REGION Network 1: Khi thang máy ở tầng 1
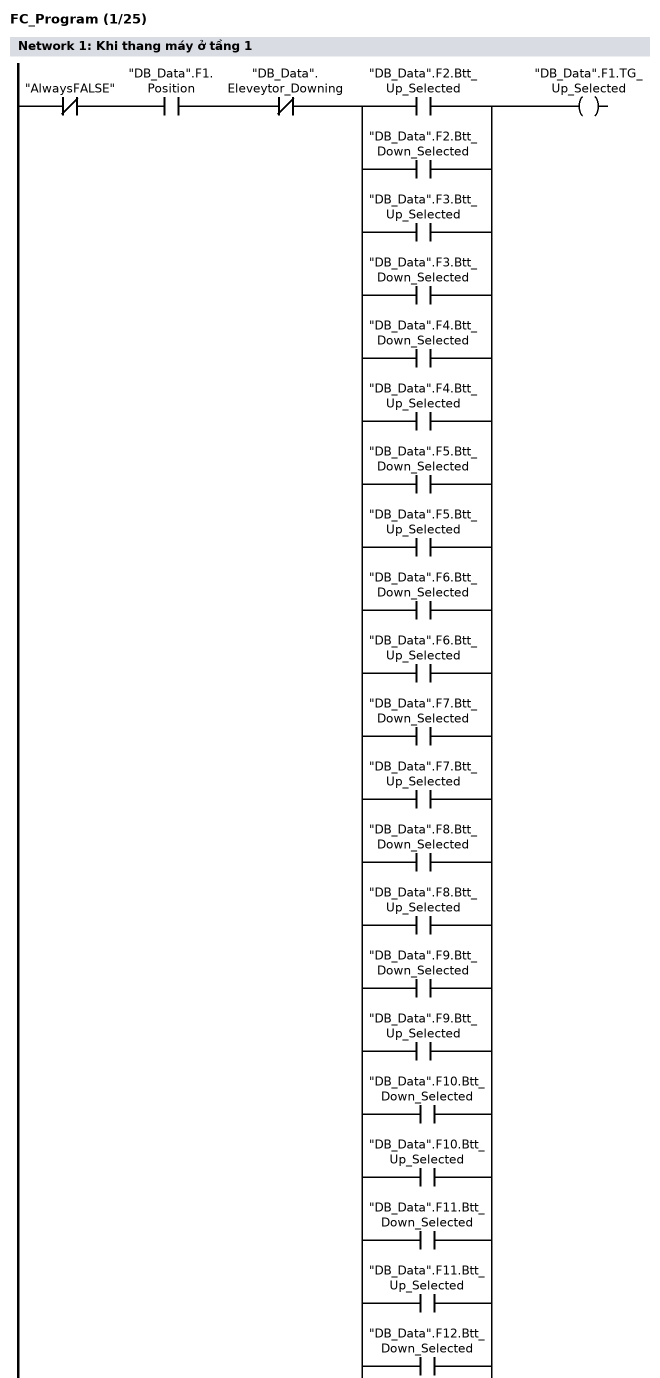
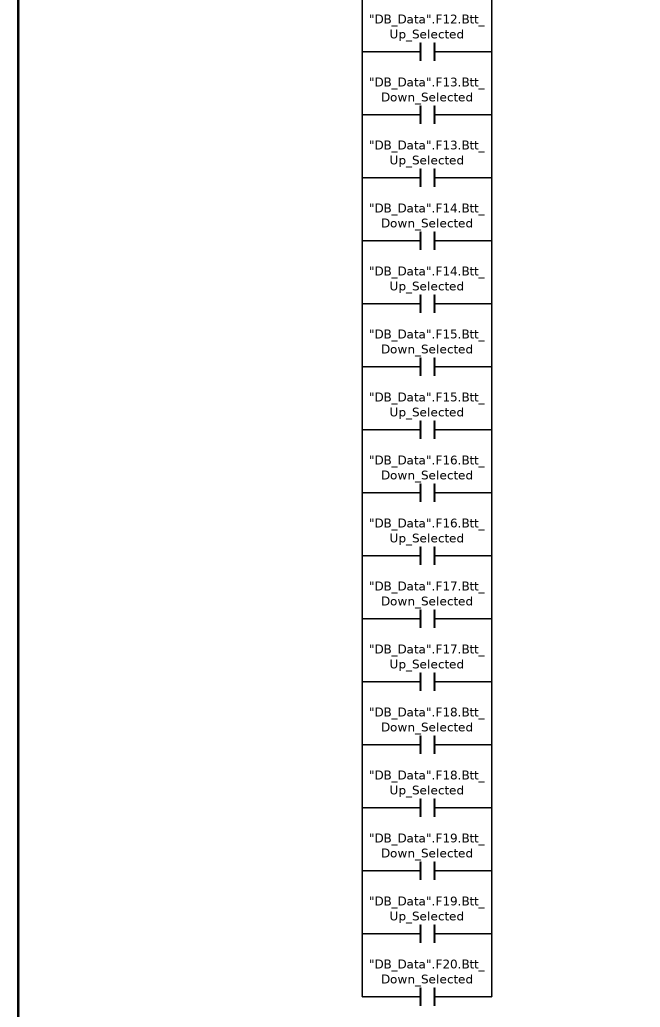
   RUNG wire#powerrail
      I_Contact( "AlwaysFALSE" )
      Contact( "DB_Data".F1.Position )
      I_Contact( "DB_Data".Eleveytor_Downing )
      wire#w1
      Contact( "DB_Data".F2.Btt_Up_Selected )
      wire#w2
      Coil( "DB_Data".F1.TG_Up_Selected )
   END_RUNG
   RUNG wire#w1
      Contact( "DB_Data".F2.Btt_Down_Selected )
   END_RUNG wire#w2
   RUNG wire#w1
      Contact( "DB_Data".F3.Btt_Up_Selected )
   END_RUNG wire#w2
   RUNG wire#w1
      Contact( "DB_Data".F3.Btt_Down_Selected )
   END_RUNG wire#w2
   RUNG wire#w1
      Contact( "DB_Data".F4.Btt_Down_Selected )
   END_RUNG wire#w2
   RUNG wire#w1
      Contact( "DB_Data".F4.Btt_Up_Selected )
   END_RUNG wire#w2
   RUNG wire#w1
      Contact( "DB_Data".F5.Btt_Down_Selected )
   END_RUNG wire#w2
   RUNG wire#w1
      Contact( "DB_Data".F5.Btt_Up_Selected )
   END_RUNG wire#w2
   RUNG wire#w1
      Contact( "DB_Data".F6.Btt_Down_Selected )
   END_RUNG wire#w2
   RUNG wire#w1
      Contact( "DB_Data".F6.Btt_Up_Selected )
   END_RUNG wire#w2
   RUNG wire#w1
      Contact( "DB_Data".F7.Btt_Down_Selected )
   END_RUNG wire#w2
   RUNG wire#w1
      Contact( "DB_Data".F7.Btt_Up_Selected )
   END_RUNG wire#w2
   RUNG wire#w1
      Contact( "DB_Data".F8.Btt_Down_Selected )
   END_RUNG wire#w2
   RUNG wire#w1
      Contact( "DB_Data".F8.Btt_Up_Selected )
   END_RUNG wire#w2
   RUNG wire#w1
      Contact( "DB_Data".F9.Btt_Down_Selected )
   END_RUNG wire#w2
   RUNG wire#w1
      Contact( "DB_Data".F9.Btt_Up_Selected )
   END_RUNG wire#w2
   RUNG wire#w1
      Contact( "DB_Data".F10.Btt_Down_Selected )
   END_RUNG wire#w2
   RUNG wire#w1
      Contact( "DB_Data".F10.Btt_Up_Selected )
   END_RUNG wire#w2
   RUNG wire#w1
      Contact( "DB_Data".F11.Btt_Down_Selected )
   END_RUNG wire#w2
   RUNG wire#w1
      Contact( "DB_Data".F11.Btt_Up_Selected )
   END_RUNG wire#w2
   RUNG wire#w1
      Contact( "DB_Data".F12.Btt_Down_Selected )
   END_RUNG wire#w2
   RUNG wire#w1
      Contact( "DB_Data".F12.Btt_Up_Selected )
   END_RUNG wire#w2
   RUNG wire#w1
      Contact( "DB_Data".F13.Btt_Down_Selected )
   END_RUNG wire#w2
   RUNG wire#w1
      Contact( "DB_Data".F13.Btt_Up_Selected )
   END_RUNG wire#w2
   RUNG wire#w1
      Contact( "DB_Data".F14.Btt_Down_Selected )
   END_RUNG wire#w2
   RUNG wire#w1
      Contact( "DB_Data".F14.Btt_Up_Selected )
   END_RUNG wire#w2
   RUNG wire#w1
      Contact( "DB_Data".F15.Btt_Down_Selected )
   END_RUNG wire#w2
   RUNG wire#w1
      Contact( "DB_Data".F15.Btt_Up_Selected )
   END_RUNG wire#w2
   RUNG wire#w1
      Contact( "DB_Data".F16.Btt_Down_Selected )
   END_RUNG wire#w2
   RUNG wire#w1
      Contact( "DB_Data".F16.Btt_Up_Selected )
   END_RUNG wire#w2
   RUNG wire#w1
      Contact( "DB_Data".F17.Btt_Down_Selected )
   END_RUNG wire#w2
   RUNG wire#w1
      Contact( "DB_Data".F17.Btt_Up_Selected )
   END_RUNG wire#w2
   RUNG wire#w1
      Contact( "DB_Data".F18.Btt_Down_Selected )
   END_RUNG wire#w2
   RUNG wire#w1
      Contact( "DB_Data".F18.Btt_Up_Selected )
   END_RUNG wire#w2
   RUNG wire#w1
      Contact( "DB_Data".F19.Btt_Down_Selected )
   END_RUNG wire#w2
   RUNG wire#w1
      Contact( "DB_Data".F19.Btt_Up_Selected )
   END_RUNG wire#w2
   RUNG wire#w1
      Contact( "DB_Data".F20.Btt_Down_Selected )
   END_RUNG wire#w2
   // the same network as SCL:
   "DB_Data".F1.TG_Up_Selected := NOT "AlwaysFALSE" AND "DB_Data".F1.Position AND NOT "DB_Data".Eleveytor_Downing AND ("DB_Data".F2.Btt_Up_Selected OR "DB_Data".F2.Btt_Down_Selected OR "DB_Data".F3.Btt_Up_Selected OR "DB_Data".F3.Btt_Down_Selected OR "DB_Data".F4.Btt_Down_Selected OR "DB_Data".F4.Btt_Up_Selected OR "DB_Data".F5.Btt_Down_Selected OR "DB_Data".F5.Btt_Up_Selected OR "DB_Data".F6.Btt_Down_Selected OR "DB_Data".F6.Btt_Up_Selected OR "DB_Data".F7.Btt_Down_Selected OR "DB_Data".F7.Btt_Up_Selected OR "DB_Data".F8.Btt_Down_Selected OR "DB_Data".F8.Btt_Up_Selected OR "DB_Data".F9.Btt_Down_Selected OR "DB_Data".F9.Btt_Up_Selected OR "DB_Data".F10.Btt_Down_Selected OR "DB_Data".F10.Btt_Up_Selected OR "DB_Data".F11.Btt_Down_Selected OR "DB_Data".F11.Btt_Up_Selected OR "DB_Data".F12.Btt_Down_Selected OR "DB_Data".F12.Btt_Up_Selected OR "DB_Data".F13.Btt_Down_Selected OR "DB_Data".F13.Btt_Up_Selected OR "DB_Data".F14.Btt_Down_Selected OR "DB_Data".F14.Btt_Up_Selected OR "DB_Data".F15.Btt_Down_Selected OR "DB_Data".F15.Btt_Up_Selected OR "DB_Data".F16.Btt_Down_Selected OR "DB_Data".F16.Btt_Up_Selected OR "DB_Data".F17.Btt_Down_Selected OR "DB_Data".F17.Btt_Up_Selected OR "DB_Data".F18.Btt_Down_Selected OR "DB_Data".F18.Btt_Up_Selected OR "DB_Data".F19.Btt_Down_Selected OR "DB_Data".F19.Btt_Up_Selected OR "DB_Data".F20.Btt_Down_Selected);
END_REGION

REGION Network 2: Khi thang máy ở tầng 2
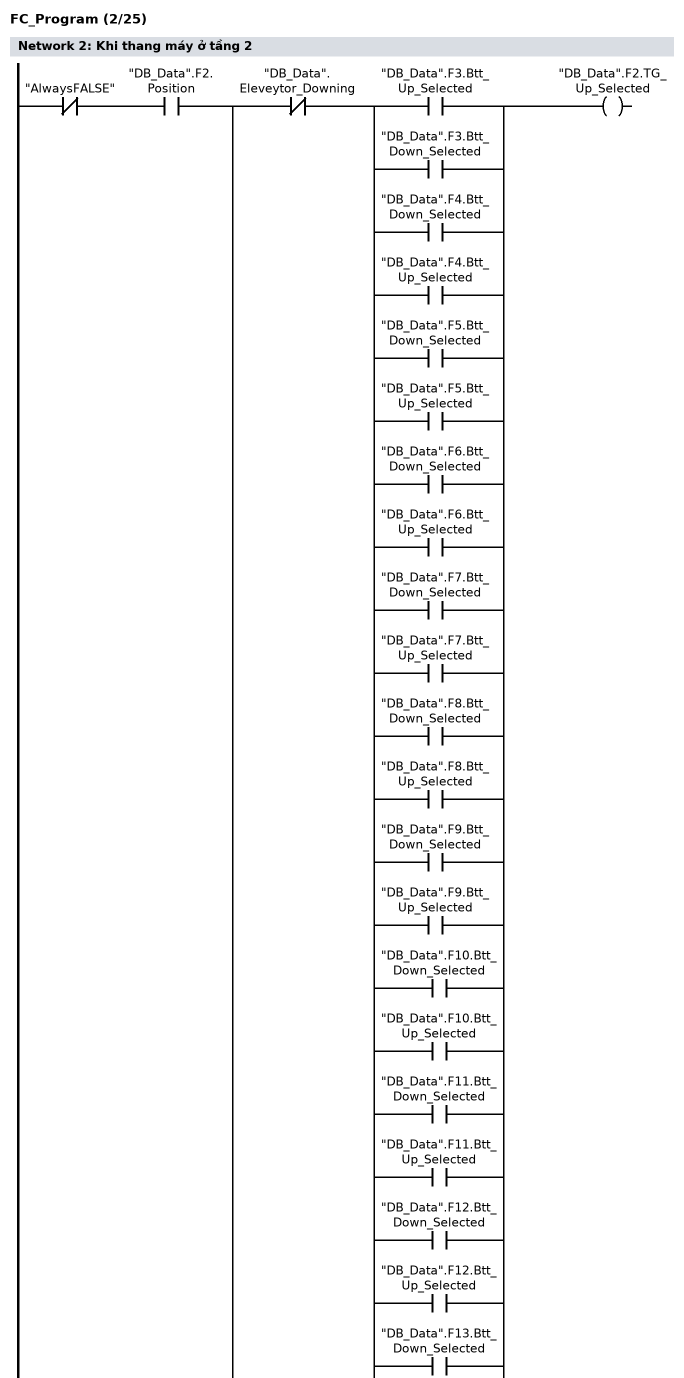
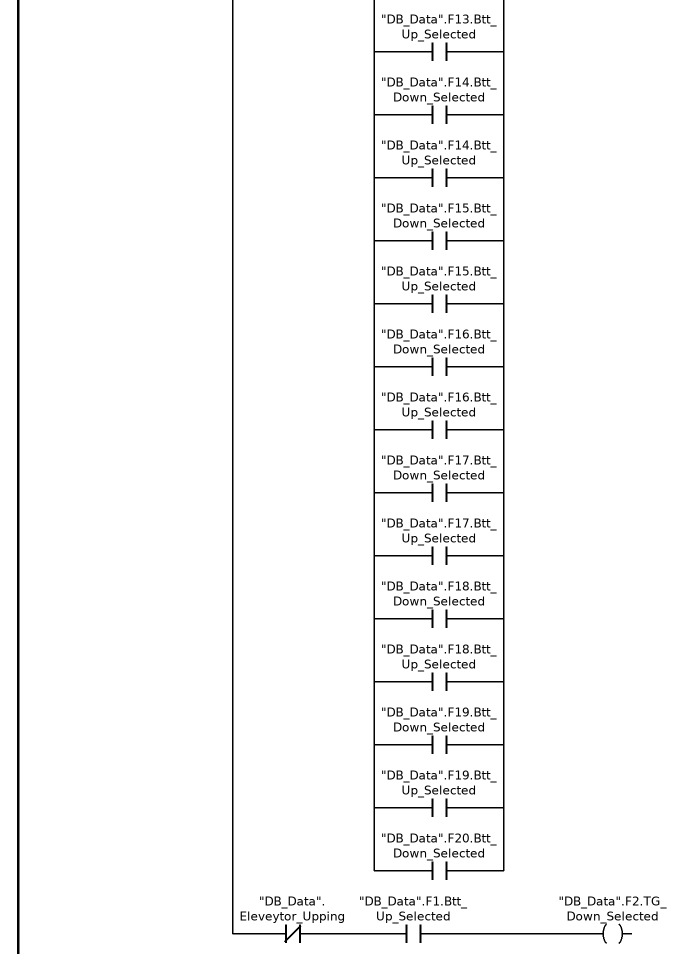
   RUNG wire#powerrail
      I_Contact( "AlwaysFALSE" )
      Contact( "DB_Data".F2.Position )
      wire#w1
      I_Contact( "DB_Data".Eleveytor_Downing )
      wire#w2
      Contact( "DB_Data".F3.Btt_Up_Selected )
      wire#w3
      Coil( "DB_Data".F2.TG_Up_Selected )
   END_RUNG
   RUNG wire#w2
      Contact( "DB_Data".F3.Btt_Down_Selected )
   END_RUNG wire#w3
   RUNG wire#w2
      Contact( "DB_Data".F4.Btt_Down_Selected )
   END_RUNG wire#w3
   RUNG wire#w2
      Contact( "DB_Data".F4.Btt_Up_Selected )
   END_RUNG wire#w3
   RUNG wire#w2
      Contact( "DB_Data".F5.Btt_Down_Selected )
   END_RUNG wire#w3
   RUNG wire#w2
      Contact( "DB_Data".F5.Btt_Up_Selected )
   END_RUNG wire#w3
   RUNG wire#w2
      Contact( "DB_Data".F6.Btt_Down_Selected )
   END_RUNG wire#w3
   RUNG wire#w2
      Contact( "DB_Data".F6.Btt_Up_Selected )
   END_RUNG wire#w3
   RUNG wire#w2
      Contact( "DB_Data".F7.Btt_Down_Selected )
   END_RUNG wire#w3
   RUNG wire#w2
      Contact( "DB_Data".F7.Btt_Up_Selected )
   END_RUNG wire#w3
   RUNG wire#w2
      Contact( "DB_Data".F8.Btt_Down_Selected )
   END_RUNG wire#w3
   RUNG wire#w2
      Contact( "DB_Data".F8.Btt_Up_Selected )
   END_RUNG wire#w3
   RUNG wire#w2
      Contact( "DB_Data".F9.Btt_Down_Selected )
   END_RUNG wire#w3
   RUNG wire#w2
      Contact( "DB_Data".F9.Btt_Up_Selected )
   END_RUNG wire#w3
   RUNG wire#w2
      Contact( "DB_Data".F10.Btt_Down_Selected )
   END_RUNG wire#w3
   RUNG wire#w2
      Contact( "DB_Data".F10.Btt_Up_Selected )
   END_RUNG wire#w3
   RUNG wire#w2
      Contact( "DB_Data".F11.Btt_Down_Selected )
   END_RUNG wire#w3
   RUNG wire#w2
      Contact( "DB_Data".F11.Btt_Up_Selected )
   END_RUNG wire#w3
   RUNG wire#w2
      Contact( "DB_Data".F12.Btt_Down_Selected )
   END_RUNG wire#w3
   RUNG wire#w2
      Contact( "DB_Data".F12.Btt_Up_Selected )
   END_RUNG wire#w3
   RUNG wire#w2
      Contact( "DB_Data".F13.Btt_Down_Selected )
   END_RUNG wire#w3
   RUNG wire#w2
      Contact( "DB_Data".F13.Btt_Up_Selected )
   END_RUNG wire#w3
   RUNG wire#w2
      Contact( "DB_Data".F14.Btt_Down_Selected )
   END_RUNG wire#w3
   RUNG wire#w2
      Contact( "DB_Data".F14.Btt_Up_Selected )
   END_RUNG wire#w3
   RUNG wire#w2
      Contact( "DB_Data".F15.Btt_Down_Selected )
   END_RUNG wire#w3
   RUNG wire#w2
      Contact( "DB_Data".F15.Btt_Up_Selected )
   END_RUNG wire#w3
   RUNG wire#w2
      Contact( "DB_Data".F16.Btt_Down_Selected )
   END_RUNG wire#w3
   RUNG wire#w2
      Contact( "DB_Data".F16.Btt_Up_Selected )
   END_RUNG wire#w3
   RUNG wire#w2
      Contact( "DB_Data".F17.Btt_Down_Selected )
   END_RUNG wire#w3
   RUNG wire#w2
      Contact( "DB_Data".F17.Btt_Up_Selected )
   END_RUNG wire#w3
   RUNG wire#w2
      Contact( "DB_Data".F18.Btt_Down_Selected )
   END_RUNG wire#w3
   RUNG wire#w2
      Contact( "DB_Data".F18.Btt_Up_Selected )
   END_RUNG wire#w3
   RUNG wire#w2
      Contact( "DB_Data".F19.Btt_Down_Selected )
   END_RUNG wire#w3
   RUNG wire#w2
      Contact( "DB_Data".F19.Btt_Up_Selected )
   END_RUNG wire#w3
   RUNG wire#w2
      Contact( "DB_Data".F20.Btt_Down_Selected )
   END_RUNG wire#w3
   RUNG wire#w1
      I_Contact( "DB_Data".Eleveytor_Upping )
      Contact( "DB_Data".F1.Btt_Up_Selected )
      Coil( "DB_Data".F2.TG_Down_Selected )
   END_RUNG
   // the same network as SCL:
   #_w1 := NOT "AlwaysFALSE" AND "DB_Data".F2.Position;
   "DB_Data".F2.TG_Up_Selected := #_w1 AND NOT "DB_Data".Eleveytor_Downing AND ("DB_Data".F3.Btt_Up_Selected OR "DB_Data".F3.Btt_Down_Selected OR "DB_Data".F4.Btt_Down_Selected OR "DB_Data".F4.Btt_Up_Selected OR "DB_Data".F5.Btt_Down_Selected OR "DB_Data".F5.Btt_Up_Selected OR "DB_Data".F6.Btt_Down_Selected OR "DB_Data".F6.Btt_Up_Selected OR "DB_Data".F7.Btt_Down_Selected OR "DB_Data".F7.Btt_Up_Selected OR "DB_Data".F8.Btt_Down_Selected OR "DB_Data".F8.Btt_Up_Selected OR "DB_Data".F9.Btt_Down_Selected OR "DB_Data".F9.Btt_Up_Selected OR "DB_Data".F10.Btt_Down_Selected OR "DB_Data".F10.Btt_Up_Selected OR "DB_Data".F11.Btt_Down_Selected OR "DB_Data".F11.Btt_Up_Selected OR "DB_Data".F12.Btt_Down_Selected OR "DB_Data".F12.Btt_Up_Selected OR "DB_Data".F13.Btt_Down_Selected OR "DB_Data".F13.Btt_Up_Selected OR "DB_Data".F14.Btt_Down_Selected OR "DB_Data".F14.Btt_Up_Selected OR "DB_Data".F15.Btt_Down_Selected OR "DB_Data".F15.Btt_Up_Selected OR "DB_Data".F16.Btt_Down_Selected OR "DB_Data".F16.Btt_Up_Selected OR "DB_Data".F17.Btt_Down_Selected OR "DB_Data".F17.Btt_Up_Selected OR "DB_Data".F18.Btt_Down_Selected OR "DB_Data".F18.Btt_Up_Selected OR "DB_Data".F19.Btt_Down_Selected OR "DB_Data".F19.Btt_Up_Selected OR "DB_Data".F20.Btt_Down_Selected);
   "DB_Data".F2.TG_Down_Selected := #_w1 AND NOT "DB_Data".Eleveytor_Upping AND "DB_Data".F1.Btt_Up_Selected;
END_REGION

REGION Network 3: Khi thang máy ở tầng 3
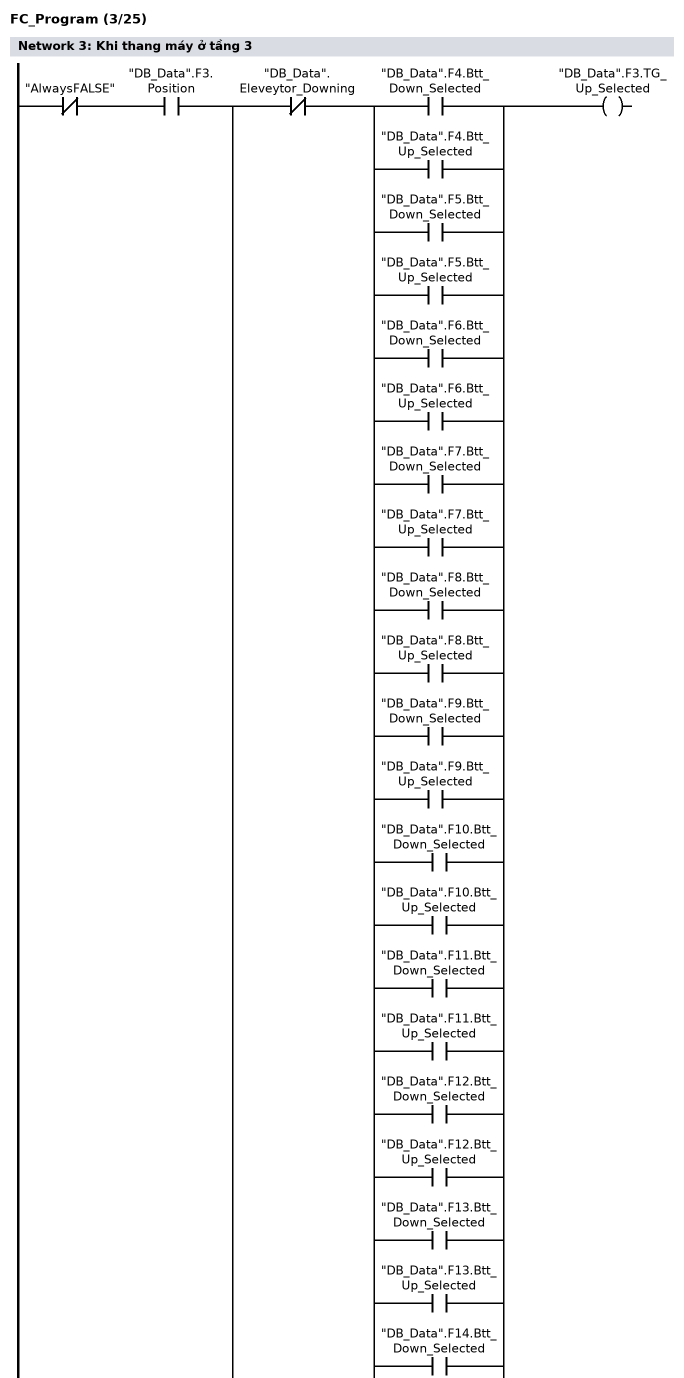
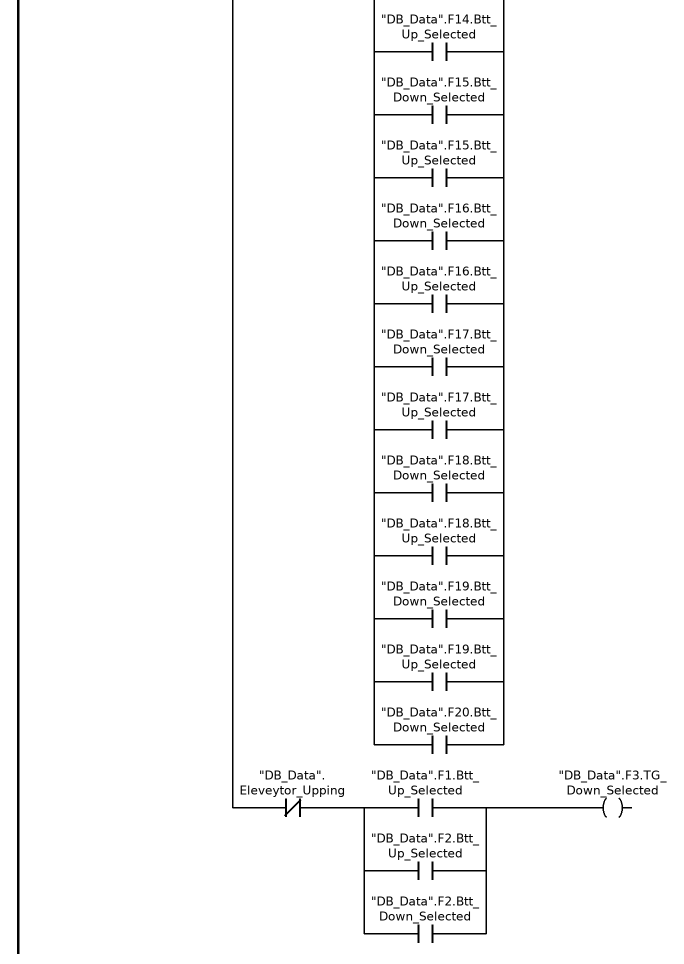
   RUNG wire#powerrail
      I_Contact( "AlwaysFALSE" )
      Contact( "DB_Data".F3.Position )
      wire#w1
      I_Contact( "DB_Data".Eleveytor_Downing )
      wire#w2
      Contact( "DB_Data".F4.Btt_Down_Selected )
      wire#w3
      Coil( "DB_Data".F3.TG_Up_Selected )
   END_RUNG
   RUNG wire#w2
      Contact( "DB_Data".F4.Btt_Up_Selected )
   END_RUNG wire#w3
   RUNG wire#w2
      Contact( "DB_Data".F5.Btt_Down_Selected )
   END_RUNG wire#w3
   RUNG wire#w2
      Contact( "DB_Data".F5.Btt_Up_Selected )
   END_RUNG wire#w3
   RUNG wire#w2
      Contact( "DB_Data".F6.Btt_Down_Selected )
   END_RUNG wire#w3
   RUNG wire#w2
      Contact( "DB_Data".F6.Btt_Up_Selected )
   END_RUNG wire#w3
   RUNG wire#w2
      Contact( "DB_Data".F7.Btt_Down_Selected )
   END_RUNG wire#w3
   RUNG wire#w2
      Contact( "DB_Data".F7.Btt_Up_Selected )
   END_RUNG wire#w3
   RUNG wire#w2
      Contact( "DB_Data".F8.Btt_Down_Selected )
   END_RUNG wire#w3
   RUNG wire#w2
      Contact( "DB_Data".F8.Btt_Up_Selected )
   END_RUNG wire#w3
   RUNG wire#w2
      Contact( "DB_Data".F9.Btt_Down_Selected )
   END_RUNG wire#w3
   RUNG wire#w2
      Contact( "DB_Data".F9.Btt_Up_Selected )
   END_RUNG wire#w3
   RUNG wire#w2
      Contact( "DB_Data".F10.Btt_Down_Selected )
   END_RUNG wire#w3
   RUNG wire#w2
      Contact( "DB_Data".F10.Btt_Up_Selected )
   END_RUNG wire#w3
   RUNG wire#w2
      Contact( "DB_Data".F11.Btt_Down_Selected )
   END_RUNG wire#w3
   RUNG wire#w2
      Contact( "DB_Data".F11.Btt_Up_Selected )
   END_RUNG wire#w3
   RUNG wire#w2
      Contact( "DB_Data".F12.Btt_Down_Selected )
   END_RUNG wire#w3
   RUNG wire#w2
      Contact( "DB_Data".F12.Btt_Up_Selected )
   END_RUNG wire#w3
   RUNG wire#w2
      Contact( "DB_Data".F13.Btt_Down_Selected )
   END_RUNG wire#w3
   RUNG wire#w2
      Contact( "DB_Data".F13.Btt_Up_Selected )
   END_RUNG wire#w3
   RUNG wire#w2
      Contact( "DB_Data".F14.Btt_Down_Selected )
   END_RUNG wire#w3
   RUNG wire#w2
      Contact( "DB_Data".F14.Btt_Up_Selected )
   END_RUNG wire#w3
   RUNG wire#w2
      Contact( "DB_Data".F15.Btt_Down_Selected )
   END_RUNG wire#w3
   RUNG wire#w2
      Contact( "DB_Data".F15.Btt_Up_Selected )
   END_RUNG wire#w3
   RUNG wire#w2
      Contact( "DB_Data".F16.Btt_Down_Selected )
   END_RUNG wire#w3
   RUNG wire#w2
      Contact( "DB_Data".F16.Btt_Up_Selected )
   END_RUNG wire#w3
   RUNG wire#w2
      Contact( "DB_Data".F17.Btt_Down_Selected )
   END_RUNG wire#w3
   RUNG wire#w2
      Contact( "DB_Data".F17.Btt_Up_Selected )
   END_RUNG wire#w3
   RUNG wire#w2
      Contact( "DB_Data".F18.Btt_Down_Selected )
   END_RUNG wire#w3
   RUNG wire#w2
      Contact( "DB_Data".F18.Btt_Up_Selected )
   END_RUNG wire#w3
   RUNG wire#w2
      Contact( "DB_Data".F19.Btt_Down_Selected )
   END_RUNG wire#w3
   RUNG wire#w2
      Contact( "DB_Data".F19.Btt_Up_Selected )
   END_RUNG wire#w3
   RUNG wire#w2
      Contact( "DB_Data".F20.Btt_Down_Selected )
   END_RUNG wire#w3
   RUNG wire#w1
      I_Contact( "DB_Data".Eleveytor_Upping )
      wire#w4
      Contact( "DB_Data".F1.Btt_Up_Selected )
      wire#w5
      Coil( "DB_Data".F3.TG_Down_Selected )
   END_RUNG
   RUNG wire#w4
      Contact( "DB_Data".F2.Btt_Up_Selected )
   END_RUNG wire#w5
   RUNG wire#w4
      Contact( "DB_Data".F2.Btt_Down_Selected )
   END_RUNG wire#w5
   // the same network as SCL:
   #_w1 := NOT "AlwaysFALSE" AND "DB_Data".F3.Position;
   "DB_Data".F3.TG_Up_Selected := #_w1 AND NOT "DB_Data".Eleveytor_Downing AND ("DB_Data".F4.Btt_Down_Selected OR "DB_Data".F4.Btt_Up_Selected OR "DB_Data".F5.Btt_Down_Selected OR "DB_Data".F5.Btt_Up_Selected OR "DB_Data".F6.Btt_Down_Selected OR "DB_Data".F6.Btt_Up_Selected OR "DB_Data".F7.Btt_Down_Selected OR "DB_Data".F7.Btt_Up_Selected OR "DB_Data".F8.Btt_Down_Selected OR "DB_Data".F8.Btt_Up_Selected OR "DB_Data".F9.Btt_Down_Selected OR "DB_Data".F9.Btt_Up_Selected OR "DB_Data".F10.Btt_Down_Selected OR "DB_Data".F10.Btt_Up_Selected OR "DB_Data".F11.Btt_Down_Selected OR "DB_Data".F11.Btt_Up_Selected OR "DB_Data".F12.Btt_Down_Selected OR "DB_Data".F12.Btt_Up_Selected OR "DB_Data".F13.Btt_Down_Selected OR "DB_Data".F13.Btt_Up_Selected OR "DB_Data".F14.Btt_Down_Selected OR "DB_Data".F14.Btt_Up_Selected OR "DB_Data".F15.Btt_Down_Selected OR "DB_Data".F15.Btt_Up_Selected OR "DB_Data".F16.Btt_Down_Selected OR "DB_Data".F16.Btt_Up_Selected OR "DB_Data".F17.Btt_Down_Selected OR "DB_Data".F17.Btt_Up_Selected OR "DB_Data".F18.Btt_Down_Selected OR "DB_Data".F18.Btt_Up_Selected OR "DB_Data".F19.Btt_Down_Selected OR "DB_Data".F19.Btt_Up_Selected OR "DB_Data".F20.Btt_Down_Selected);
   "DB_Data".F3.TG_Down_Selected := #_w1 AND NOT "DB_Data".Eleveytor_Upping AND ("DB_Data".F1.Btt_Up_Selected OR "DB_Data".F2.Btt_Up_Selected OR "DB_Data".F2.Btt_Down_Selected);
END_REGION

REGION Network 4: Khi thang máy ở tầng 4
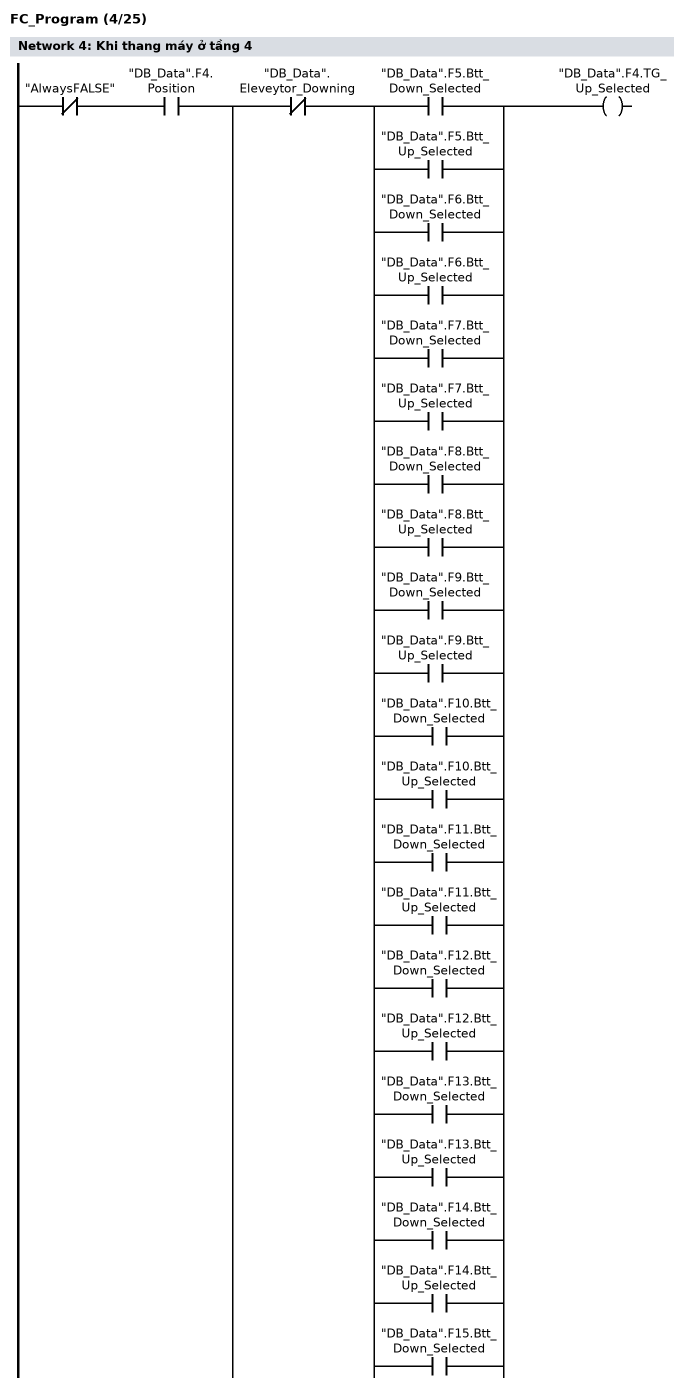
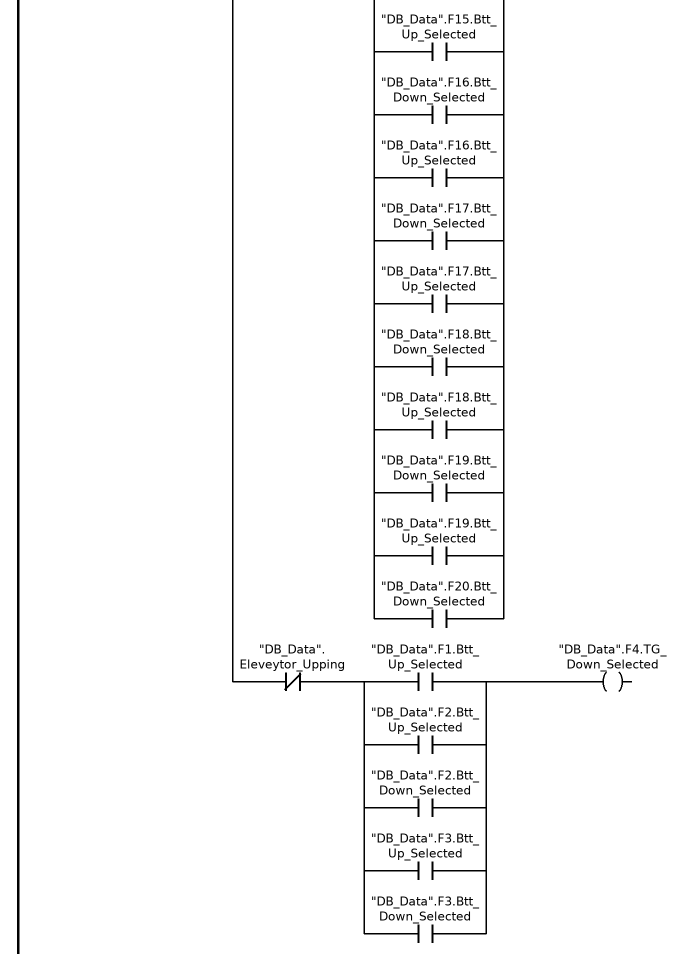
   RUNG wire#powerrail
      I_Contact( "AlwaysFALSE" )
      Contact( "DB_Data".F4.Position )
      wire#w1
      I_Contact( "DB_Data".Eleveytor_Downing )
      wire#w2
      Contact( "DB_Data".F5.Btt_Down_Selected )
      wire#w3
      Coil( "DB_Data".F4.TG_Up_Selected )
   END_RUNG
   RUNG wire#w2
      Contact( "DB_Data".F5.Btt_Up_Selected )
   END_RUNG wire#w3
   RUNG wire#w2
      Contact( "DB_Data".F6.Btt_Down_Selected )
   END_RUNG wire#w3
   RUNG wire#w2
      Contact( "DB_Data".F6.Btt_Up_Selected )
   END_RUNG wire#w3
   RUNG wire#w2
      Contact( "DB_Data".F7.Btt_Down_Selected )
   END_RUNG wire#w3
   RUNG wire#w2
      Contact( "DB_Data".F7.Btt_Up_Selected )
   END_RUNG wire#w3
   RUNG wire#w2
      Contact( "DB_Data".F8.Btt_Down_Selected )
   END_RUNG wire#w3
   RUNG wire#w2
      Contact( "DB_Data".F8.Btt_Up_Selected )
   END_RUNG wire#w3
   RUNG wire#w2
      Contact( "DB_Data".F9.Btt_Down_Selected )
   END_RUNG wire#w3
   RUNG wire#w2
      Contact( "DB_Data".F9.Btt_Up_Selected )
   END_RUNG wire#w3
   RUNG wire#w2
      Contact( "DB_Data".F10.Btt_Down_Selected )
   END_RUNG wire#w3
   RUNG wire#w2
      Contact( "DB_Data".F10.Btt_Up_Selected )
   END_RUNG wire#w3
   RUNG wire#w2
      Contact( "DB_Data".F11.Btt_Down_Selected )
   END_RUNG wire#w3
   RUNG wire#w2
      Contact( "DB_Data".F11.Btt_Up_Selected )
   END_RUNG wire#w3
   RUNG wire#w2
      Contact( "DB_Data".F12.Btt_Down_Selected )
   END_RUNG wire#w3
   RUNG wire#w2
      Contact( "DB_Data".F12.Btt_Up_Selected )
   END_RUNG wire#w3
   RUNG wire#w2
      Contact( "DB_Data".F13.Btt_Down_Selected )
   END_RUNG wire#w3
   RUNG wire#w2
      Contact( "DB_Data".F13.Btt_Up_Selected )
   END_RUNG wire#w3
   RUNG wire#w2
      Contact( "DB_Data".F14.Btt_Down_Selected )
   END_RUNG wire#w3
   RUNG wire#w2
      Contact( "DB_Data".F14.Btt_Up_Selected )
   END_RUNG wire#w3
   RUNG wire#w2
      Contact( "DB_Data".F15.Btt_Down_Selected )
   END_RUNG wire#w3
   RUNG wire#w2
      Contact( "DB_Data".F15.Btt_Up_Selected )
   END_RUNG wire#w3
   RUNG wire#w2
      Contact( "DB_Data".F16.Btt_Down_Selected )
   END_RUNG wire#w3
   RUNG wire#w2
      Contact( "DB_Data".F16.Btt_Up_Selected )
   END_RUNG wire#w3
   RUNG wire#w2
      Contact( "DB_Data".F17.Btt_Down_Selected )
   END_RUNG wire#w3
   RUNG wire#w2
      Contact( "DB_Data".F17.Btt_Up_Selected )
   END_RUNG wire#w3
   RUNG wire#w2
      Contact( "DB_Data".F18.Btt_Down_Selected )
   END_RUNG wire#w3
   RUNG wire#w2
      Contact( "DB_Data".F18.Btt_Up_Selected )
   END_RUNG wire#w3
   RUNG wire#w2
      Contact( "DB_Data".F19.Btt_Down_Selected )
   END_RUNG wire#w3
   RUNG wire#w2
      Contact( "DB_Data".F19.Btt_Up_Selected )
   END_RUNG wire#w3
   RUNG wire#w2
      Contact( "DB_Data".F20.Btt_Down_Selected )
   END_RUNG wire#w3
   RUNG wire#w1
      I_Contact( "DB_Data".Eleveytor_Upping )
      wire#w4
      Contact( "DB_Data".F1.Btt_Up_Selected )
      wire#w5
      Coil( "DB_Data".F4.TG_Down_Selected )
   END_RUNG
   RUNG wire#w4
      Contact( "DB_Data".F2.Btt_Up_Selected )
   END_RUNG wire#w5
   RUNG wire#w4
      Contact( "DB_Data".F2.Btt_Down_Selected )
   END_RUNG wire#w5
   RUNG wire#w4
      Contact( "DB_Data".F3.Btt_Up_Selected )
   END_RUNG wire#w5
   RUNG wire#w4
      Contact( "DB_Data".F3.Btt_Down_Selected )
   END_RUNG wire#w5
   // the same network as SCL:
   #_w1 := NOT "AlwaysFALSE" AND "DB_Data".F4.Position;
   "DB_Data".F4.TG_Up_Selected := #_w1 AND NOT "DB_Data".Eleveytor_Downing AND ("DB_Data".F5.Btt_Down_Selected OR "DB_Data".F5.Btt_Up_Selected OR "DB_Data".F6.Btt_Down_Selected OR "DB_Data".F6.Btt_Up_Selected OR "DB_Data".F7.Btt_Down_Selected OR "DB_Data".F7.Btt_Up_Selected OR "DB_Data".F8.Btt_Down_Selected OR "DB_Data".F8.Btt_Up_Selected OR "DB_Data".F9.Btt_Down_Selected OR "DB_Data".F9.Btt_Up_Selected OR "DB_Data".F10.Btt_Down_Selected OR "DB_Data".F10.Btt_Up_Selected OR "DB_Data".F11.Btt_Down_Selected OR "DB_Data".F11.Btt_Up_Selected OR "DB_Data".F12.Btt_Down_Selected OR "DB_Data".F12.Btt_Up_Selected OR "DB_Data".F13.Btt_Down_Selected OR "DB_Data".F13.Btt_Up_Selected OR "DB_Data".F14.Btt_Down_Selected OR "DB_Data".F14.Btt_Up_Selected OR "DB_Data".F15.Btt_Down_Selected OR "DB_Data".F15.Btt_Up_Selected OR "DB_Data".F16.Btt_Down_Selected OR "DB_Data".F16.Btt_Up_Selected OR "DB_Data".F17.Btt_Down_Selected OR "DB_Data".F17.Btt_Up_Selected OR "DB_Data".F18.Btt_Down_Selected OR "DB_Data".F18.Btt_Up_Selected OR "DB_Data".F19.Btt_Down_Selected OR "DB_Data".F19.Btt_Up_Selected OR "DB_Data".F20.Btt_Down_Selected);
   "DB_Data".F4.TG_Down_Selected := #_w1 AND NOT "DB_Data".Eleveytor_Upping AND ("DB_Data".F1.Btt_Up_Selected OR "DB_Data".F2.Btt_Up_Selected OR "DB_Data".F2.Btt_Down_Selected OR "DB_Data".F3.Btt_Up_Selected OR "DB_Data".F3.Btt_Down_Selected);
END_REGION

REGION Network 5: Khi thang máy ở tầng 5
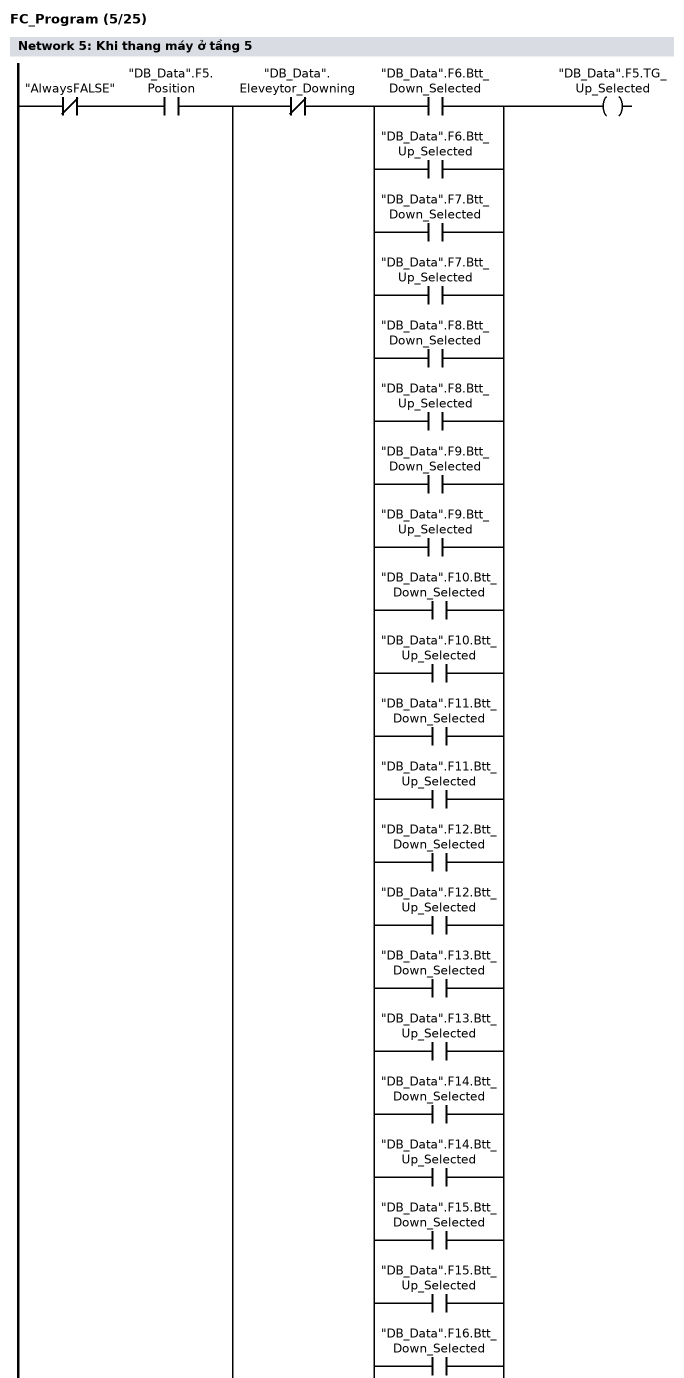
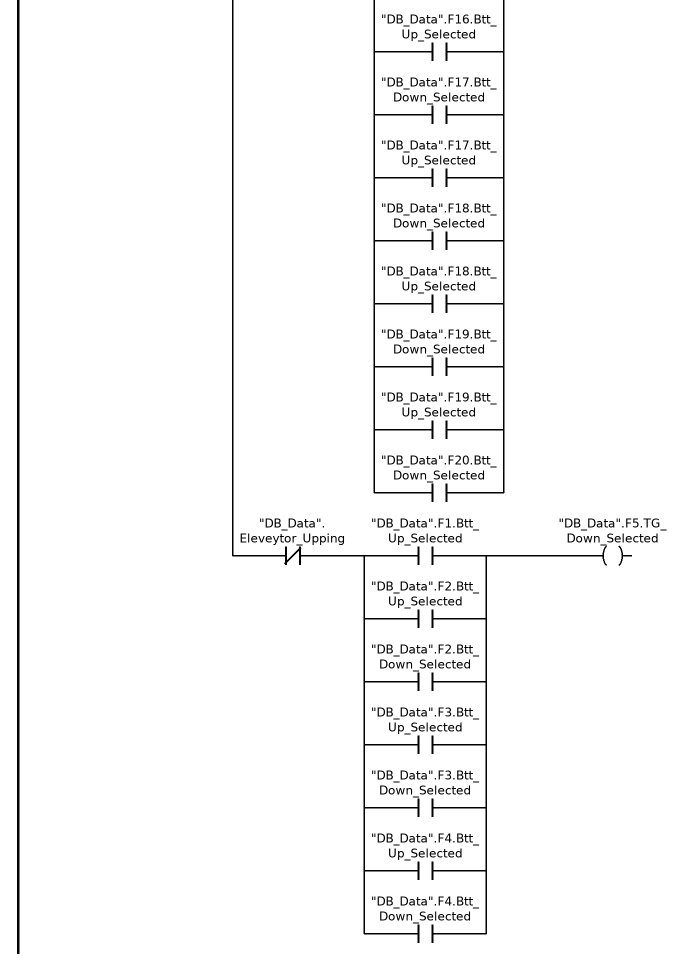
   RUNG wire#powerrail
      I_Contact( "AlwaysFALSE" )
      Contact( "DB_Data".F5.Position )
      wire#w1
      I_Contact( "DB_Data".Eleveytor_Downing )
      wire#w2
      Contact( "DB_Data".F6.Btt_Down_Selected )
      wire#w3
      Coil( "DB_Data".F5.TG_Up_Selected )
   END_RUNG
   RUNG wire#w2
      Contact( "DB_Data".F6.Btt_Up_Selected )
   END_RUNG wire#w3
   RUNG wire#w2
      Contact( "DB_Data".F7.Btt_Down_Selected )
   END_RUNG wire#w3
   RUNG wire#w2
      Contact( "DB_Data".F7.Btt_Up_Selected )
   END_RUNG wire#w3
   RUNG wire#w2
      Contact( "DB_Data".F8.Btt_Down_Selected )
   END_RUNG wire#w3
   RUNG wire#w2
      Contact( "DB_Data".F8.Btt_Up_Selected )
   END_RUNG wire#w3
   RUNG wire#w2
      Contact( "DB_Data".F9.Btt_Down_Selected )
   END_RUNG wire#w3
   RUNG wire#w2
      Contact( "DB_Data".F9.Btt_Up_Selected )
   END_RUNG wire#w3
   RUNG wire#w2
      Contact( "DB_Data".F10.Btt_Down_Selected )
   END_RUNG wire#w3
   RUNG wire#w2
      Contact( "DB_Data".F10.Btt_Up_Selected )
   END_RUNG wire#w3
   RUNG wire#w2
      Contact( "DB_Data".F11.Btt_Down_Selected )
   END_RUNG wire#w3
   RUNG wire#w2
      Contact( "DB_Data".F11.Btt_Up_Selected )
   END_RUNG wire#w3
   RUNG wire#w2
      Contact( "DB_Data".F12.Btt_Down_Selected )
   END_RUNG wire#w3
   RUNG wire#w2
      Contact( "DB_Data".F12.Btt_Up_Selected )
   END_RUNG wire#w3
   RUNG wire#w2
      Contact( "DB_Data".F13.Btt_Down_Selected )
   END_RUNG wire#w3
   RUNG wire#w2
      Contact( "DB_Data".F13.Btt_Up_Selected )
   END_RUNG wire#w3
   RUNG wire#w2
      Contact( "DB_Data".F14.Btt_Down_Selected )
   END_RUNG wire#w3
   RUNG wire#w2
      Contact( "DB_Data".F14.Btt_Up_Selected )
   END_RUNG wire#w3
   RUNG wire#w2
      Contact( "DB_Data".F15.Btt_Down_Selected )
   END_RUNG wire#w3
   RUNG wire#w2
      Contact( "DB_Data".F15.Btt_Up_Selected )
   END_RUNG wire#w3
   RUNG wire#w2
      Contact( "DB_Data".F16.Btt_Down_Selected )
   END_RUNG wire#w3
   RUNG wire#w2
      Contact( "DB_Data".F16.Btt_Up_Selected )
   END_RUNG wire#w3
   RUNG wire#w2
      Contact( "DB_Data".F17.Btt_Down_Selected )
   END_RUNG wire#w3
   RUNG wire#w2
      Contact( "DB_Data".F17.Btt_Up_Selected )
   END_RUNG wire#w3
   RUNG wire#w2
      Contact( "DB_Data".F18.Btt_Down_Selected )
   END_RUNG wire#w3
   RUNG wire#w2
      Contact( "DB_Data".F18.Btt_Up_Selected )
   END_RUNG wire#w3
   RUNG wire#w2
      Contact( "DB_Data".F19.Btt_Down_Selected )
   END_RUNG wire#w3
   RUNG wire#w2
      Contact( "DB_Data".F19.Btt_Up_Selected )
   END_RUNG wire#w3
   RUNG wire#w2
      Contact( "DB_Data".F20.Btt_Down_Selected )
   END_RUNG wire#w3
   RUNG wire#w1
      I_Contact( "DB_Data".Eleveytor_Upping )
      wire#w4
      Contact( "DB_Data".F1.Btt_Up_Selected )
      wire#w5
      Coil( "DB_Data".F5.TG_Down_Selected )
   END_RUNG
   RUNG wire#w4
      Contact( "DB_Data".F2.Btt_Up_Selected )
   END_RUNG wire#w5
   RUNG wire#w4
      Contact( "DB_Data".F2.Btt_Down_Selected )
   END_RUNG wire#w5
   RUNG wire#w4
      Contact( "DB_Data".F3.Btt_Up_Selected )
   END_RUNG wire#w5
   RUNG wire#w4
      Contact( "DB_Data".F3.Btt_Down_Selected )
   END_RUNG wire#w5
   RUNG wire#w4
      Contact( "DB_Data".F4.Btt_Up_Selected )
   END_RUNG wire#w5
   RUNG wire#w4
      Contact( "DB_Data".F4.Btt_Down_Selected )
   END_RUNG wire#w5
   // the same network as SCL:
   #_w1 := NOT "AlwaysFALSE" AND "DB_Data".F5.Position;
   "DB_Data".F5.TG_Up_Selected := #_w1 AND NOT "DB_Data".Eleveytor_Downing AND ("DB_Data".F6.Btt_Down_Selected OR "DB_Data".F6.Btt_Up_Selected OR "DB_Data".F7.Btt_Down_Selected OR "DB_Data".F7.Btt_Up_Selected OR "DB_Data".F8.Btt_Down_Selected OR "DB_Data".F8.Btt_Up_Selected OR "DB_Data".F9.Btt_Down_Selected OR "DB_Data".F9.Btt_Up_Selected OR "DB_Data".F10.Btt_Down_Selected OR "DB_Data".F10.Btt_Up_Selected OR "DB_Data".F11.Btt_Down_Selected OR "DB_Data".F11.Btt_Up_Selected OR "DB_Data".F12.Btt_Down_Selected OR "DB_Data".F12.Btt_Up_Selected OR "DB_Data".F13.Btt_Down_Selected OR "DB_Data".F13.Btt_Up_Selected OR "DB_Data".F14.Btt_Down_Selected OR "DB_Data".F14.Btt_Up_Selected OR "DB_Data".F15.Btt_Down_Selected OR "DB_Data".F15.Btt_Up_Selected OR "DB_Data".F16.Btt_Down_Selected OR "DB_Data".F16.Btt_Up_Selected OR "DB_Data".F17.Btt_Down_Selected OR "DB_Data".F17.Btt_Up_Selected OR "DB_Data".F18.Btt_Down_Selected OR "DB_Data".F18.Btt_Up_Selected OR "DB_Data".F19.Btt_Down_Selected OR "DB_Data".F19.Btt_Up_Selected OR "DB_Data".F20.Btt_Down_Selected);
   "DB_Data".F5.TG_Down_Selected := #_w1 AND NOT "DB_Data".Eleveytor_Upping AND ("DB_Data".F1.Btt_Up_Selected OR "DB_Data".F2.Btt_Up_Selected OR "DB_Data".F2.Btt_Down_Selected OR "DB_Data".F3.Btt_Up_Selected OR "DB_Data".F3.Btt_Down_Selected OR "DB_Data".F4.Btt_Up_Selected OR "DB_Data".F4.Btt_Down_Selected);
END_REGION

REGION Network 6: Khi thang máy ở tầng 6
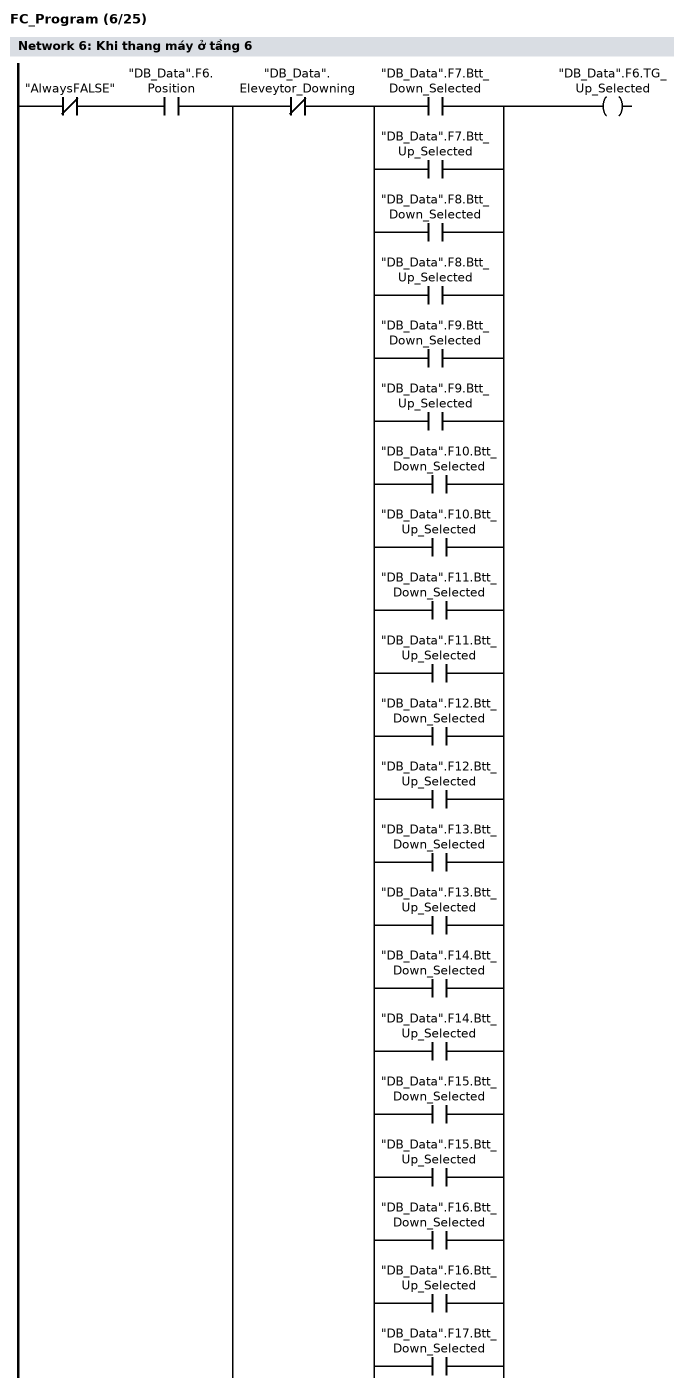
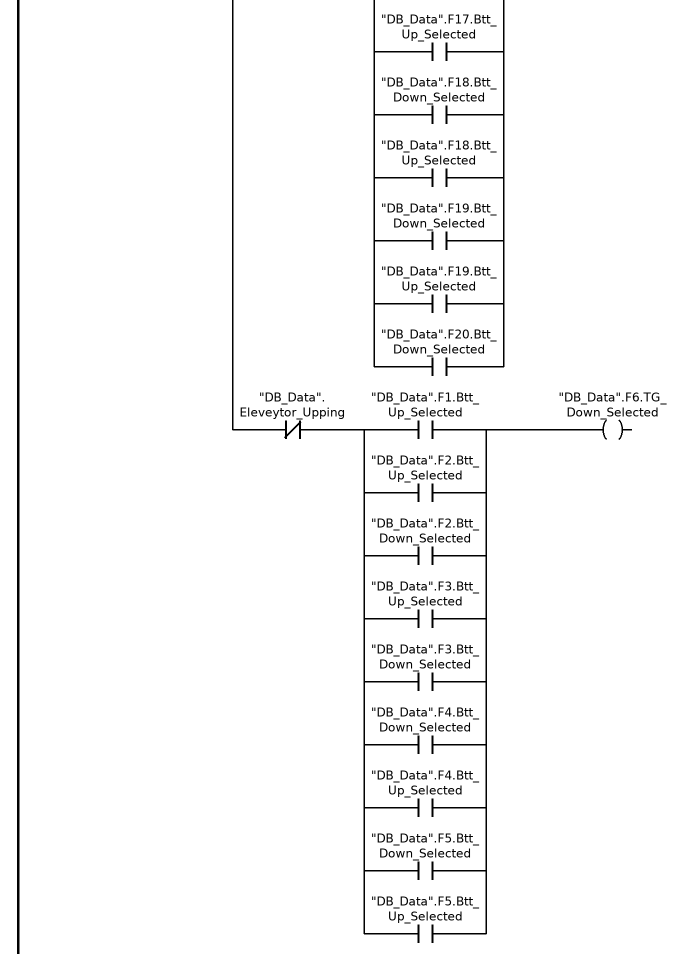
   RUNG wire#powerrail
      I_Contact( "AlwaysFALSE" )
      Contact( "DB_Data".F6.Position )
      wire#w1
      I_Contact( "DB_Data".Eleveytor_Downing )
      wire#w2
      Contact( "DB_Data".F7.Btt_Down_Selected )
      wire#w3
      Coil( "DB_Data".F6.TG_Up_Selected )
   END_RUNG
   RUNG wire#w2
      Contact( "DB_Data".F7.Btt_Up_Selected )
   END_RUNG wire#w3
   RUNG wire#w2
      Contact( "DB_Data".F8.Btt_Down_Selected )
   END_RUNG wire#w3
   RUNG wire#w2
      Contact( "DB_Data".F8.Btt_Up_Selected )
   END_RUNG wire#w3
   RUNG wire#w2
      Contact( "DB_Data".F9.Btt_Down_Selected )
   END_RUNG wire#w3
   RUNG wire#w2
      Contact( "DB_Data".F9.Btt_Up_Selected )
   END_RUNG wire#w3
   RUNG wire#w2
      Contact( "DB_Data".F10.Btt_Down_Selected )
   END_RUNG wire#w3
   RUNG wire#w2
      Contact( "DB_Data".F10.Btt_Up_Selected )
   END_RUNG wire#w3
   RUNG wire#w2
      Contact( "DB_Data".F11.Btt_Down_Selected )
   END_RUNG wire#w3
   RUNG wire#w2
      Contact( "DB_Data".F11.Btt_Up_Selected )
   END_RUNG wire#w3
   RUNG wire#w2
      Contact( "DB_Data".F12.Btt_Down_Selected )
   END_RUNG wire#w3
   RUNG wire#w2
      Contact( "DB_Data".F12.Btt_Up_Selected )
   END_RUNG wire#w3
   RUNG wire#w2
      Contact( "DB_Data".F13.Btt_Down_Selected )
   END_RUNG wire#w3
   RUNG wire#w2
      Contact( "DB_Data".F13.Btt_Up_Selected )
   END_RUNG wire#w3
   RUNG wire#w2
      Contact( "DB_Data".F14.Btt_Down_Selected )
   END_RUNG wire#w3
   RUNG wire#w2
      Contact( "DB_Data".F14.Btt_Up_Selected )
   END_RUNG wire#w3
   RUNG wire#w2
      Contact( "DB_Data".F15.Btt_Down_Selected )
   END_RUNG wire#w3
   RUNG wire#w2
      Contact( "DB_Data".F15.Btt_Up_Selected )
   END_RUNG wire#w3
   RUNG wire#w2
      Contact( "DB_Data".F16.Btt_Down_Selected )
   END_RUNG wire#w3
   RUNG wire#w2
      Contact( "DB_Data".F16.Btt_Up_Selected )
   END_RUNG wire#w3
   RUNG wire#w2
      Contact( "DB_Data".F17.Btt_Down_Selected )
   END_RUNG wire#w3
   RUNG wire#w2
      Contact( "DB_Data".F17.Btt_Up_Selected )
   END_RUNG wire#w3
   RUNG wire#w2
      Contact( "DB_Data".F18.Btt_Down_Selected )
   END_RUNG wire#w3
   RUNG wire#w2
      Contact( "DB_Data".F18.Btt_Up_Selected )
   END_RUNG wire#w3
   RUNG wire#w2
      Contact( "DB_Data".F19.Btt_Down_Selected )
   END_RUNG wire#w3
   RUNG wire#w2
      Contact( "DB_Data".F19.Btt_Up_Selected )
   END_RUNG wire#w3
   RUNG wire#w2
      Contact( "DB_Data".F20.Btt_Down_Selected )
   END_RUNG wire#w3
   RUNG wire#w1
      I_Contact( "DB_Data".Eleveytor_Upping )
      wire#w4
      Contact( "DB_Data".F1.Btt_Up_Selected )
      wire#w5
      Coil( "DB_Data".F6.TG_Down_Selected )
   END_RUNG
   RUNG wire#w4
      Contact( "DB_Data".F2.Btt_Up_Selected )
   END_RUNG wire#w5
   RUNG wire#w4
      Contact( "DB_Data".F2.Btt_Down_Selected )
   END_RUNG wire#w5
   RUNG wire#w4
      Contact( "DB_Data".F3.Btt_Up_Selected )
   END_RUNG wire#w5
   RUNG wire#w4
      Contact( "DB_Data".F3.Btt_Down_Selected )
   END_RUNG wire#w5
   RUNG wire#w4
      Contact( "DB_Data".F4.Btt_Down_Selected )
   END_RUNG wire#w5
   RUNG wire#w4
      Contact( "DB_Data".F4.Btt_Up_Selected )
   END_RUNG wire#w5
   RUNG wire#w4
      Contact( "DB_Data".F5.Btt_Down_Selected )
   END_RUNG wire#w5
   RUNG wire#w4
      Contact( "DB_Data".F5.Btt_Up_Selected )
   END_RUNG wire#w5
   // the same network as SCL:
   #_w1 := NOT "AlwaysFALSE" AND "DB_Data".F6.Position;
   "DB_Data".F6.TG_Up_Selected := #_w1 AND NOT "DB_Data".Eleveytor_Downing AND ("DB_Data".F7.Btt_Down_Selected OR "DB_Data".F7.Btt_Up_Selected OR "DB_Data".F8.Btt_Down_Selected OR "DB_Data".F8.Btt_Up_Selected OR "DB_Data".F9.Btt_Down_Selected OR "DB_Data".F9.Btt_Up_Selected OR "DB_Data".F10.Btt_Down_Selected OR "DB_Data".F10.Btt_Up_Selected OR "DB_Data".F11.Btt_Down_Selected OR "DB_Data".F11.Btt_Up_Selected OR "DB_Data".F12.Btt_Down_Selected OR "DB_Data".F12.Btt_Up_Selected OR "DB_Data".F13.Btt_Down_Selected OR "DB_Data".F13.Btt_Up_Selected OR "DB_Data".F14.Btt_Down_Selected OR "DB_Data".F14.Btt_Up_Selected OR "DB_Data".F15.Btt_Down_Selected OR "DB_Data".F15.Btt_Up_Selected OR "DB_Data".F16.Btt_Down_Selected OR "DB_Data".F16.Btt_Up_Selected OR "DB_Data".F17.Btt_Down_Selected OR "DB_Data".F17.Btt_Up_Selected OR "DB_Data".F18.Btt_Down_Selected OR "DB_Data".F18.Btt_Up_Selected OR "DB_Data".F19.Btt_Down_Selected OR "DB_Data".F19.Btt_Up_Selected OR "DB_Data".F20.Btt_Down_Selected);
   "DB_Data".F6.TG_Down_Selected := #_w1 AND NOT "DB_Data".Eleveytor_Upping AND ("DB_Data".F1.Btt_Up_Selected OR "DB_Data".F2.Btt_Up_Selected OR "DB_Data".F2.Btt_Down_Selected OR "DB_Data".F3.Btt_Up_Selected OR "DB_Data".F3.Btt_Down_Selected OR "DB_Data".F4.Btt_Down_Selected OR "DB_Data".F4.Btt_Up_Selected OR "DB_Data".F5.Btt_Down_Selected OR "DB_Data".F5.Btt_Up_Selected);
END_REGION

REGION Network 7: Khi thang máy ở tầng 7
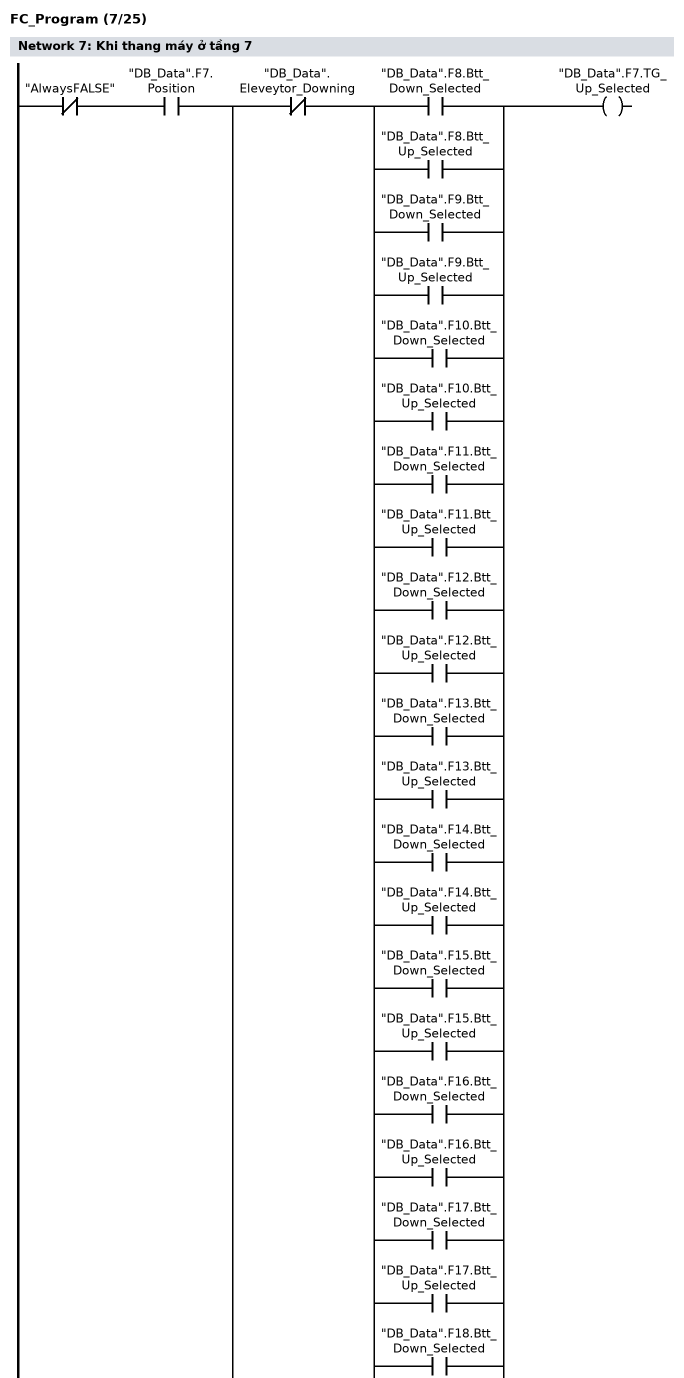
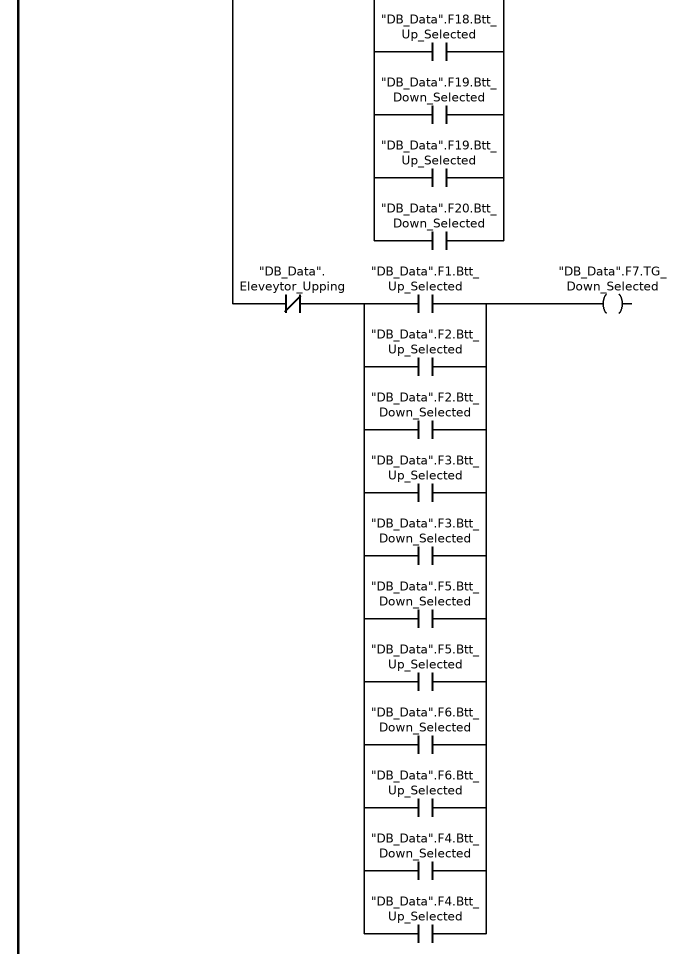
   RUNG wire#powerrail
      I_Contact( "AlwaysFALSE" )
      Contact( "DB_Data".F7.Position )
      wire#w1
      I_Contact( "DB_Data".Eleveytor_Downing )
      wire#w2
      Contact( "DB_Data".F8.Btt_Down_Selected )
      wire#w3
      Coil( "DB_Data".F7.TG_Up_Selected )
   END_RUNG
   RUNG wire#w2
      Contact( "DB_Data".F8.Btt_Up_Selected )
   END_RUNG wire#w3
   RUNG wire#w2
      Contact( "DB_Data".F9.Btt_Down_Selected )
   END_RUNG wire#w3
   RUNG wire#w2
      Contact( "DB_Data".F9.Btt_Up_Selected )
   END_RUNG wire#w3
   RUNG wire#w2
      Contact( "DB_Data".F10.Btt_Down_Selected )
   END_RUNG wire#w3
   RUNG wire#w2
      Contact( "DB_Data".F10.Btt_Up_Selected )
   END_RUNG wire#w3
   RUNG wire#w2
      Contact( "DB_Data".F11.Btt_Down_Selected )
   END_RUNG wire#w3
   RUNG wire#w2
      Contact( "DB_Data".F11.Btt_Up_Selected )
   END_RUNG wire#w3
   RUNG wire#w2
      Contact( "DB_Data".F12.Btt_Down_Selected )
   END_RUNG wire#w3
   RUNG wire#w2
      Contact( "DB_Data".F12.Btt_Up_Selected )
   END_RUNG wire#w3
   RUNG wire#w2
      Contact( "DB_Data".F13.Btt_Down_Selected )
   END_RUNG wire#w3
   RUNG wire#w2
      Contact( "DB_Data".F13.Btt_Up_Selected )
   END_RUNG wire#w3
   RUNG wire#w2
      Contact( "DB_Data".F14.Btt_Down_Selected )
   END_RUNG wire#w3
   RUNG wire#w2
      Contact( "DB_Data".F14.Btt_Up_Selected )
   END_RUNG wire#w3
   RUNG wire#w2
      Contact( "DB_Data".F15.Btt_Down_Selected )
   END_RUNG wire#w3
   RUNG wire#w2
      Contact( "DB_Data".F15.Btt_Up_Selected )
   END_RUNG wire#w3
   RUNG wire#w2
      Contact( "DB_Data".F16.Btt_Down_Selected )
   END_RUNG wire#w3
   RUNG wire#w2
      Contact( "DB_Data".F16.Btt_Up_Selected )
   END_RUNG wire#w3
   RUNG wire#w2
      Contact( "DB_Data".F17.Btt_Down_Selected )
   END_RUNG wire#w3
   RUNG wire#w2
      Contact( "DB_Data".F17.Btt_Up_Selected )
   END_RUNG wire#w3
   RUNG wire#w2
      Contact( "DB_Data".F18.Btt_Down_Selected )
   END_RUNG wire#w3
   RUNG wire#w2
      Contact( "DB_Data".F18.Btt_Up_Selected )
   END_RUNG wire#w3
   RUNG wire#w2
      Contact( "DB_Data".F19.Btt_Down_Selected )
   END_RUNG wire#w3
   RUNG wire#w2
      Contact( "DB_Data".F19.Btt_Up_Selected )
   END_RUNG wire#w3
   RUNG wire#w2
      Contact( "DB_Data".F20.Btt_Down_Selected )
   END_RUNG wire#w3
   RUNG wire#w1
      I_Contact( "DB_Data".Eleveytor_Upping )
      wire#w4
      Contact( "DB_Data".F1.Btt_Up_Selected )
      wire#w5
      Coil( "DB_Data".F7.TG_Down_Selected )
   END_RUNG
   RUNG wire#w4
      Contact( "DB_Data".F2.Btt_Up_Selected )
   END_RUNG wire#w5
   RUNG wire#w4
      Contact( "DB_Data".F2.Btt_Down_Selected )
   END_RUNG wire#w5
   RUNG wire#w4
      Contact( "DB_Data".F3.Btt_Up_Selected )
   END_RUNG wire#w5
   RUNG wire#w4
      Contact( "DB_Data".F3.Btt_Down_Selected )
   END_RUNG wire#w5
   RUNG wire#w4
      Contact( "DB_Data".F5.Btt_Down_Selected )
   END_RUNG wire#w5
   RUNG wire#w4
      Contact( "DB_Data".F5.Btt_Up_Selected )
   END_RUNG wire#w5
   RUNG wire#w4
      Contact( "DB_Data".F6.Btt_Down_Selected )
   END_RUNG wire#w5
   RUNG wire#w4
      Contact( "DB_Data".F6.Btt_Up_Selected )
   END_RUNG wire#w5
   RUNG wire#w4
      Contact( "DB_Data".F4.Btt_Down_Selected )
   END_RUNG wire#w5
   RUNG wire#w4
      Contact( "DB_Data".F4.Btt_Up_Selected )
   END_RUNG wire#w5
   // the same network as SCL:
   #_w1 := NOT "AlwaysFALSE" AND "DB_Data".F7.Position;
   "DB_Data".F7.TG_Up_Selected := #_w1 AND NOT "DB_Data".Eleveytor_Downing AND ("DB_Data".F8.Btt_Down_Selected OR "DB_Data".F8.Btt_Up_Selected OR "DB_Data".F9.Btt_Down_Selected OR "DB_Data".F9.Btt_Up_Selected OR "DB_Data".F10.Btt_Down_Selected OR "DB_Data".F10.Btt_Up_Selected OR "DB_Data".F11.Btt_Down_Selected OR "DB_Data".F11.Btt_Up_Selected OR "DB_Data".F12.Btt_Down_Selected OR "DB_Data".F12.Btt_Up_Selected OR "DB_Data".F13.Btt_Down_Selected OR "DB_Data".F13.Btt_Up_Selected OR "DB_Data".F14.Btt_Down_Selected OR "DB_Data".F14.Btt_Up_Selected OR "DB_Data".F15.Btt_Down_Selected OR "DB_Data".F15.Btt_Up_Selected OR "DB_Data".F16.Btt_Down_Selected OR "DB_Data".F16.Btt_Up_Selected OR "DB_Data".F17.Btt_Down_Selected OR "DB_Data".F17.Btt_Up_Selected OR "DB_Data".F18.Btt_Down_Selected OR "DB_Data".F18.Btt_Up_Selected OR "DB_Data".F19.Btt_Down_Selected OR "DB_Data".F19.Btt_Up_Selected OR "DB_Data".F20.Btt_Down_Selected);
   "DB_Data".F7.TG_Down_Selected := #_w1 AND NOT "DB_Data".Eleveytor_Upping AND ("DB_Data".F1.Btt_Up_Selected OR "DB_Data".F2.Btt_Up_Selected OR "DB_Data".F2.Btt_Down_Selected OR "DB_Data".F3.Btt_Up_Selected OR "DB_Data".F3.Btt_Down_Selected OR "DB_Data".F5.Btt_Down_Selected OR "DB_Data".F5.Btt_Up_Selected OR "DB_Data".F6.Btt_Down_Selected OR "DB_Data".F6.Btt_Up_Selected OR "DB_Data".F4.Btt_Down_Selected OR "DB_Data".F4.Btt_Up_Selected);
END_REGION

REGION Network 8: Khi thang máy ở tầng 8
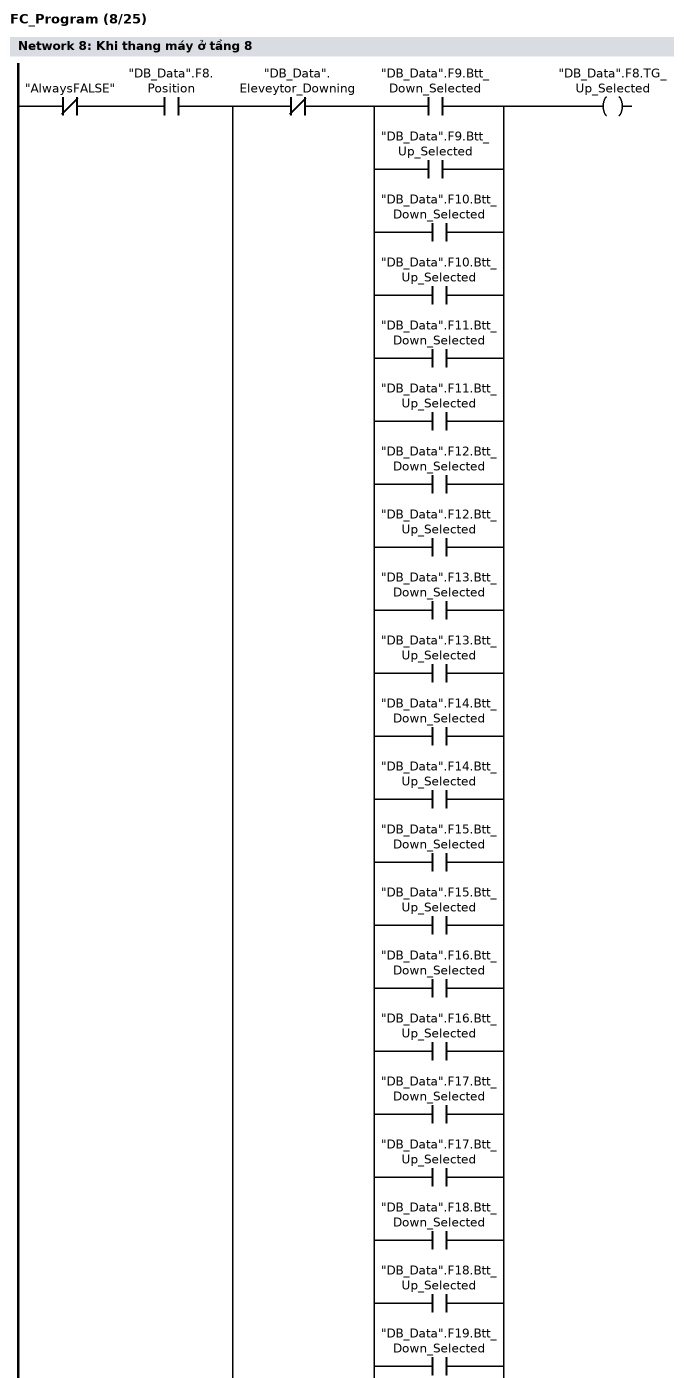
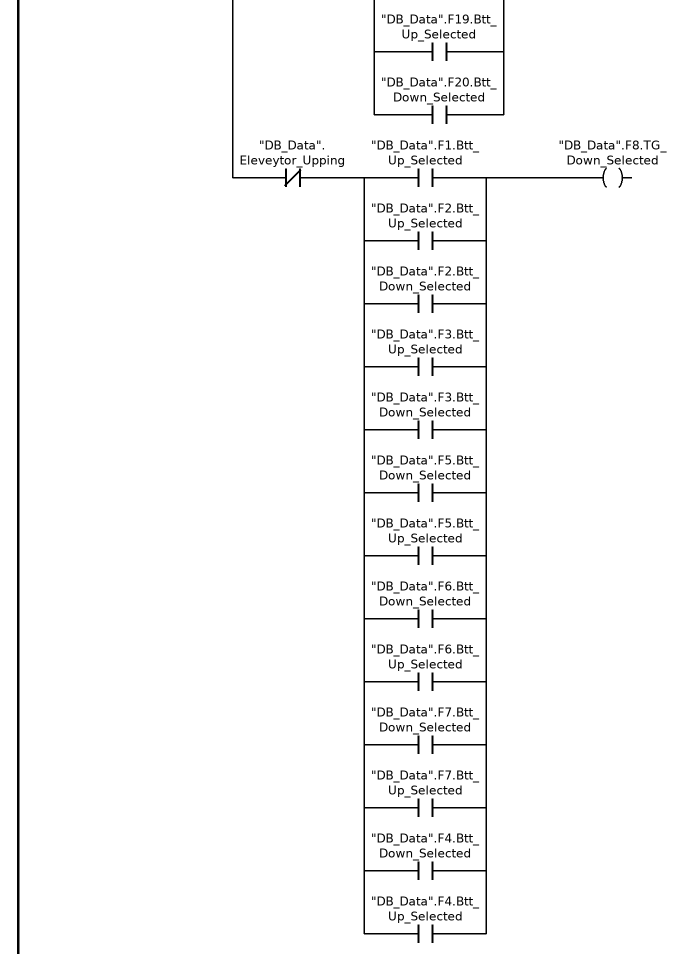
   RUNG wire#powerrail
      I_Contact( "AlwaysFALSE" )
      Contact( "DB_Data".F8.Position )
      wire#w1
      I_Contact( "DB_Data".Eleveytor_Downing )
      wire#w2
      Contact( "DB_Data".F9.Btt_Down_Selected )
      wire#w3
      Coil( "DB_Data".F8.TG_Up_Selected )
   END_RUNG
   RUNG wire#w2
      Contact( "DB_Data".F9.Btt_Up_Selected )
   END_RUNG wire#w3
   RUNG wire#w2
      Contact( "DB_Data".F10.Btt_Down_Selected )
   END_RUNG wire#w3
   RUNG wire#w2
      Contact( "DB_Data".F10.Btt_Up_Selected )
   END_RUNG wire#w3
   RUNG wire#w2
      Contact( "DB_Data".F11.Btt_Down_Selected )
   END_RUNG wire#w3
   RUNG wire#w2
      Contact( "DB_Data".F11.Btt_Up_Selected )
   END_RUNG wire#w3
   RUNG wire#w2
      Contact( "DB_Data".F12.Btt_Down_Selected )
   END_RUNG wire#w3
   RUNG wire#w2
      Contact( "DB_Data".F12.Btt_Up_Selected )
   END_RUNG wire#w3
   RUNG wire#w2
      Contact( "DB_Data".F13.Btt_Down_Selected )
   END_RUNG wire#w3
   RUNG wire#w2
      Contact( "DB_Data".F13.Btt_Up_Selected )
   END_RUNG wire#w3
   RUNG wire#w2
      Contact( "DB_Data".F14.Btt_Down_Selected )
   END_RUNG wire#w3
   RUNG wire#w2
      Contact( "DB_Data".F14.Btt_Up_Selected )
   END_RUNG wire#w3
   RUNG wire#w2
      Contact( "DB_Data".F15.Btt_Down_Selected )
   END_RUNG wire#w3
   RUNG wire#w2
      Contact( "DB_Data".F15.Btt_Up_Selected )
   END_RUNG wire#w3
   RUNG wire#w2
      Contact( "DB_Data".F16.Btt_Down_Selected )
   END_RUNG wire#w3
   RUNG wire#w2
      Contact( "DB_Data".F16.Btt_Up_Selected )
   END_RUNG wire#w3
   RUNG wire#w2
      Contact( "DB_Data".F17.Btt_Down_Selected )
   END_RUNG wire#w3
   RUNG wire#w2
      Contact( "DB_Data".F17.Btt_Up_Selected )
   END_RUNG wire#w3
   RUNG wire#w2
      Contact( "DB_Data".F18.Btt_Down_Selected )
   END_RUNG wire#w3
   RUNG wire#w2
      Contact( "DB_Data".F18.Btt_Up_Selected )
   END_RUNG wire#w3
   RUNG wire#w2
      Contact( "DB_Data".F19.Btt_Down_Selected )
   END_RUNG wire#w3
   RUNG wire#w2
      Contact( "DB_Data".F19.Btt_Up_Selected )
   END_RUNG wire#w3
   RUNG wire#w2
      Contact( "DB_Data".F20.Btt_Down_Selected )
   END_RUNG wire#w3
   RUNG wire#w1
      I_Contact( "DB_Data".Eleveytor_Upping )
      wire#w4
      Contact( "DB_Data".F1.Btt_Up_Selected )
      wire#w5
      Coil( "DB_Data".F8.TG_Down_Selected )
   END_RUNG
   RUNG wire#w4
      Contact( "DB_Data".F2.Btt_Up_Selected )
   END_RUNG wire#w5
   RUNG wire#w4
      Contact( "DB_Data".F2.Btt_Down_Selected )
   END_RUNG wire#w5
   RUNG wire#w4
      Contact( "DB_Data".F3.Btt_Up_Selected )
   END_RUNG wire#w5
   RUNG wire#w4
      Contact( "DB_Data".F3.Btt_Down_Selected )
   END_RUNG wire#w5
   RUNG wire#w4
      Contact( "DB_Data".F5.Btt_Down_Selected )
   END_RUNG wire#w5
   RUNG wire#w4
      Contact( "DB_Data".F5.Btt_Up_Selected )
   END_RUNG wire#w5
   RUNG wire#w4
      Contact( "DB_Data".F6.Btt_Down_Selected )
   END_RUNG wire#w5
   RUNG wire#w4
      Contact( "DB_Data".F6.Btt_Up_Selected )
   END_RUNG wire#w5
   RUNG wire#w4
      Contact( "DB_Data".F7.Btt_Down_Selected )
   END_RUNG wire#w5
   RUNG wire#w4
      Contact( "DB_Data".F7.Btt_Up_Selected )
   END_RUNG wire#w5
   RUNG wire#w4
      Contact( "DB_Data".F4.Btt_Down_Selected )
   END_RUNG wire#w5
   RUNG wire#w4
      Contact( "DB_Data".F4.Btt_Up_Selected )
   END_RUNG wire#w5
   // the same network as SCL:
   #_w1 := NOT "AlwaysFALSE" AND "DB_Data".F8.Position;
   "DB_Data".F8.TG_Up_Selected := #_w1 AND NOT "DB_Data".Eleveytor_Downing AND ("DB_Data".F9.Btt_Down_Selected OR "DB_Data".F9.Btt_Up_Selected OR "DB_Data".F10.Btt_Down_Selected OR "DB_Data".F10.Btt_Up_Selected OR "DB_Data".F11.Btt_Down_Selected OR "DB_Data".F11.Btt_Up_Selected OR "DB_Data".F12.Btt_Down_Selected OR "DB_Data".F12.Btt_Up_Selected OR "DB_Data".F13.Btt_Down_Selected OR "DB_Data".F13.Btt_Up_Selected OR "DB_Data".F14.Btt_Down_Selected OR "DB_Data".F14.Btt_Up_Selected OR "DB_Data".F15.Btt_Down_Selected OR "DB_Data".F15.Btt_Up_Selected OR "DB_Data".F16.Btt_Down_Selected OR "DB_Data".F16.Btt_Up_Selected OR "DB_Data".F17.Btt_Down_Selected OR "DB_Data".F17.Btt_Up_Selected OR "DB_Data".F18.Btt_Down_Selected OR "DB_Data".F18.Btt_Up_Selected OR "DB_Data".F19.Btt_Down_Selected OR "DB_Data".F19.Btt_Up_Selected OR "DB_Data".F20.Btt_Down_Selected);
   "DB_Data".F8.TG_Down_Selected := #_w1 AND NOT "DB_Data".Eleveytor_Upping AND ("DB_Data".F1.Btt_Up_Selected OR "DB_Data".F2.Btt_Up_Selected OR "DB_Data".F2.Btt_Down_Selected OR "DB_Data".F3.Btt_Up_Selected OR "DB_Data".F3.Btt_Down_Selected OR "DB_Data".F5.Btt_Down_Selected OR "DB_Data".F5.Btt_Up_Selected OR "DB_Data".F6.Btt_Down_Selected OR "DB_Data".F6.Btt_Up_Selected OR "DB_Data".F7.Btt_Down_Selected OR "DB_Data".F7.Btt_Up_Selected OR "DB_Data".F4.Btt_Down_Selected OR "DB_Data".F4.Btt_Up_Selected);
END_REGION

REGION Network 9: Khi thang máy ở tầng 9
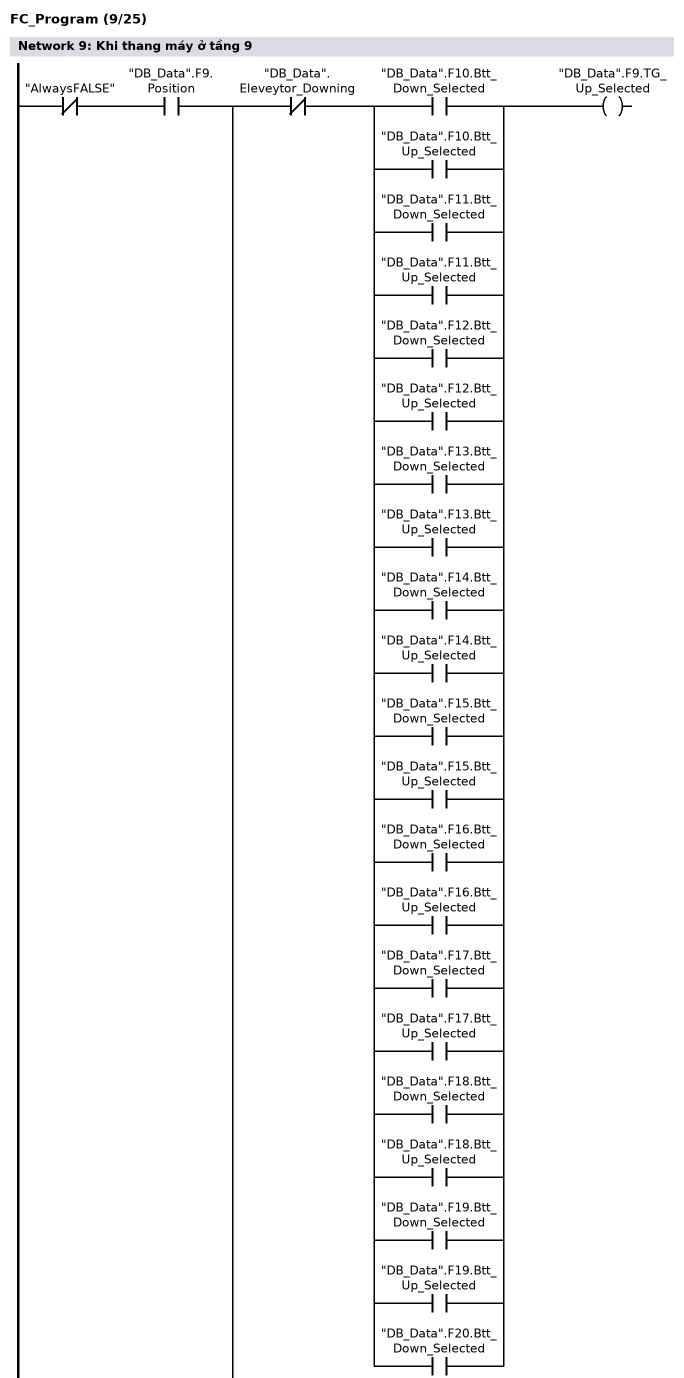
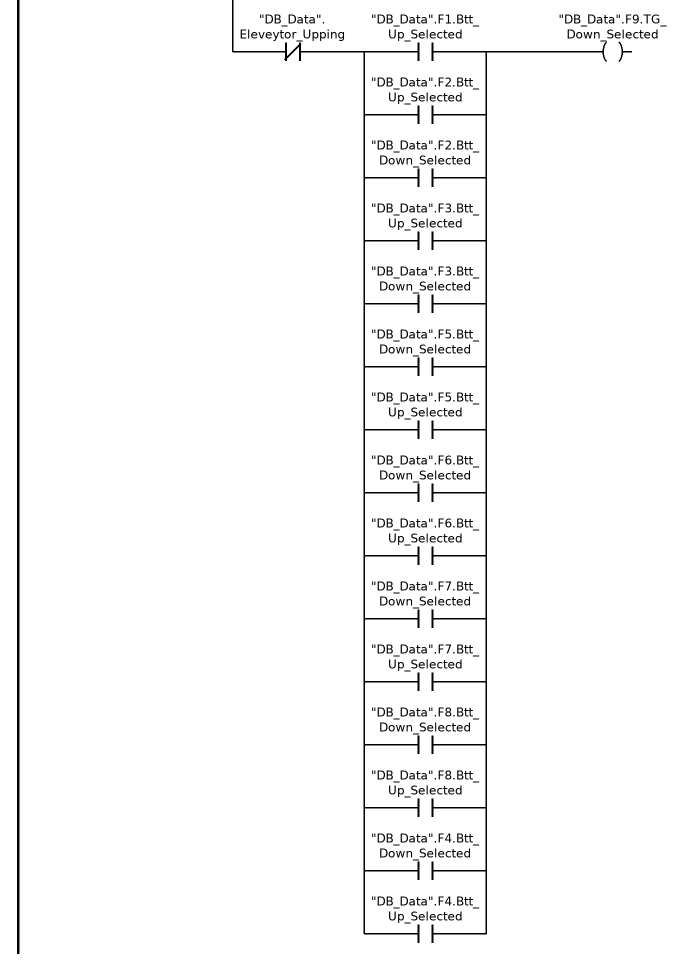
   RUNG wire#powerrail
      I_Contact( "AlwaysFALSE" )
      Contact( "DB_Data".F9.Position )
      wire#w1
      I_Contact( "DB_Data".Eleveytor_Downing )
      wire#w2
      Contact( "DB_Data".F10.Btt_Down_Selected )
      wire#w3
      Coil( "DB_Data".F9.TG_Up_Selected )
   END_RUNG
   RUNG wire#w2
      Contact( "DB_Data".F10.Btt_Up_Selected )
   END_RUNG wire#w3
   RUNG wire#w2
      Contact( "DB_Data".F11.Btt_Down_Selected )
   END_RUNG wire#w3
   RUNG wire#w2
      Contact( "DB_Data".F11.Btt_Up_Selected )
   END_RUNG wire#w3
   RUNG wire#w2
      Contact( "DB_Data".F12.Btt_Down_Selected )
   END_RUNG wire#w3
   RUNG wire#w2
      Contact( "DB_Data".F12.Btt_Up_Selected )
   END_RUNG wire#w3
   RUNG wire#w2
      Contact( "DB_Data".F13.Btt_Down_Selected )
   END_RUNG wire#w3
   RUNG wire#w2
      Contact( "DB_Data".F13.Btt_Up_Selected )
   END_RUNG wire#w3
   RUNG wire#w2
      Contact( "DB_Data".F14.Btt_Down_Selected )
   END_RUNG wire#w3
   RUNG wire#w2
      Contact( "DB_Data".F14.Btt_Up_Selected )
   END_RUNG wire#w3
   RUNG wire#w2
      Contact( "DB_Data".F15.Btt_Down_Selected )
   END_RUNG wire#w3
   RUNG wire#w2
      Contact( "DB_Data".F15.Btt_Up_Selected )
   END_RUNG wire#w3
   RUNG wire#w2
      Contact( "DB_Data".F16.Btt_Down_Selected )
   END_RUNG wire#w3
   RUNG wire#w2
      Contact( "DB_Data".F16.Btt_Up_Selected )
   END_RUNG wire#w3
   RUNG wire#w2
      Contact( "DB_Data".F17.Btt_Down_Selected )
   END_RUNG wire#w3
   RUNG wire#w2
      Contact( "DB_Data".F17.Btt_Up_Selected )
   END_RUNG wire#w3
   RUNG wire#w2
      Contact( "DB_Data".F18.Btt_Down_Selected )
   END_RUNG wire#w3
   RUNG wire#w2
      Contact( "DB_Data".F18.Btt_Up_Selected )
   END_RUNG wire#w3
   RUNG wire#w2
      Contact( "DB_Data".F19.Btt_Down_Selected )
   END_RUNG wire#w3
   RUNG wire#w2
      Contact( "DB_Data".F19.Btt_Up_Selected )
   END_RUNG wire#w3
   RUNG wire#w2
      Contact( "DB_Data".F20.Btt_Down_Selected )
   END_RUNG wire#w3
   RUNG wire#w1
      I_Contact( "DB_Data".Eleveytor_Upping )
      wire#w4
      Contact( "DB_Data".F1.Btt_Up_Selected )
      wire#w5
      Coil( "DB_Data".F9.TG_Down_Selected )
   END_RUNG
   RUNG wire#w4
      Contact( "DB_Data".F2.Btt_Up_Selected )
   END_RUNG wire#w5
   RUNG wire#w4
      Contact( "DB_Data".F2.Btt_Down_Selected )
   END_RUNG wire#w5
   RUNG wire#w4
      Contact( "DB_Data".F3.Btt_Up_Selected )
   END_RUNG wire#w5
   RUNG wire#w4
      Contact( "DB_Data".F3.Btt_Down_Selected )
   END_RUNG wire#w5
   RUNG wire#w4
      Contact( "DB_Data".F5.Btt_Down_Selected )
   END_RUNG wire#w5
   RUNG wire#w4
      Contact( "DB_Data".F5.Btt_Up_Selected )
   END_RUNG wire#w5
   RUNG wire#w4
      Contact( "DB_Data".F6.Btt_Down_Selected )
   END_RUNG wire#w5
   RUNG wire#w4
      Contact( "DB_Data".F6.Btt_Up_Selected )
   END_RUNG wire#w5
   RUNG wire#w4
      Contact( "DB_Data".F7.Btt_Down_Selected )
   END_RUNG wire#w5
   RUNG wire#w4
      Contact( "DB_Data".F7.Btt_Up_Selected )
   END_RUNG wire#w5
   RUNG wire#w4
      Contact( "DB_Data".F8.Btt_Down_Selected )
   END_RUNG wire#w5
   RUNG wire#w4
      Contact( "DB_Data".F8.Btt_Up_Selected )
   END_RUNG wire#w5
   RUNG wire#w4
      Contact( "DB_Data".F4.Btt_Down_Selected )
   END_RUNG wire#w5
   RUNG wire#w4
      Contact( "DB_Data".F4.Btt_Up_Selected )
   END_RUNG wire#w5
   // the same network as SCL:
   #_w1 := NOT "AlwaysFALSE" AND "DB_Data".F9.Position;
   "DB_Data".F9.TG_Up_Selected := #_w1 AND NOT "DB_Data".Eleveytor_Downing AND ("DB_Data".F10.Btt_Down_Selected OR "DB_Data".F10.Btt_Up_Selected OR "DB_Data".F11.Btt_Down_Selected OR "DB_Data".F11.Btt_Up_Selected OR "DB_Data".F12.Btt_Down_Selected OR "DB_Data".F12.Btt_Up_Selected OR "DB_Data".F13.Btt_Down_Selected OR "DB_Data".F13.Btt_Up_Selected OR "DB_Data".F14.Btt_Down_Selected OR "DB_Data".F14.Btt_Up_Selected OR "DB_Data".F15.Btt_Down_Selected OR "DB_Data".F15.Btt_Up_Selected OR "DB_Data".F16.Btt_Down_Selected OR "DB_Data".F16.Btt_Up_Selected OR "DB_Data".F17.Btt_Down_Selected OR "DB_Data".F17.Btt_Up_Selected OR "DB_Data".F18.Btt_Down_Selected OR "DB_Data".F18.Btt_Up_Selected OR "DB_Data".F19.Btt_Down_Selected OR "DB_Data".F19.Btt_Up_Selected OR "DB_Data".F20.Btt_Down_Selected);
   "DB_Data".F9.TG_Down_Selected := #_w1 AND NOT "DB_Data".Eleveytor_Upping AND ("DB_Data".F1.Btt_Up_Selected OR "DB_Data".F2.Btt_Up_Selected OR "DB_Data".F2.Btt_Down_Selected OR "DB_Data".F3.Btt_Up_Selected OR "DB_Data".F3.Btt_Down_Selected OR "DB_Data".F5.Btt_Down_Selected OR "DB_Data".F5.Btt_Up_Selected OR "DB_Data".F6.Btt_Down_Selected OR "DB_Data".F6.Btt_Up_Selected OR "DB_Data".F7.Btt_Down_Selected OR "DB_Data".F7.Btt_Up_Selected OR "DB_Data".F8.Btt_Down_Selected OR "DB_Data".F8.Btt_Up_Selected OR "DB_Data".F4.Btt_Down_Selected OR "DB_Data".F4.Btt_Up_Selected);
END_REGION

REGION Network 10: Khi thang máy ở tầng 10
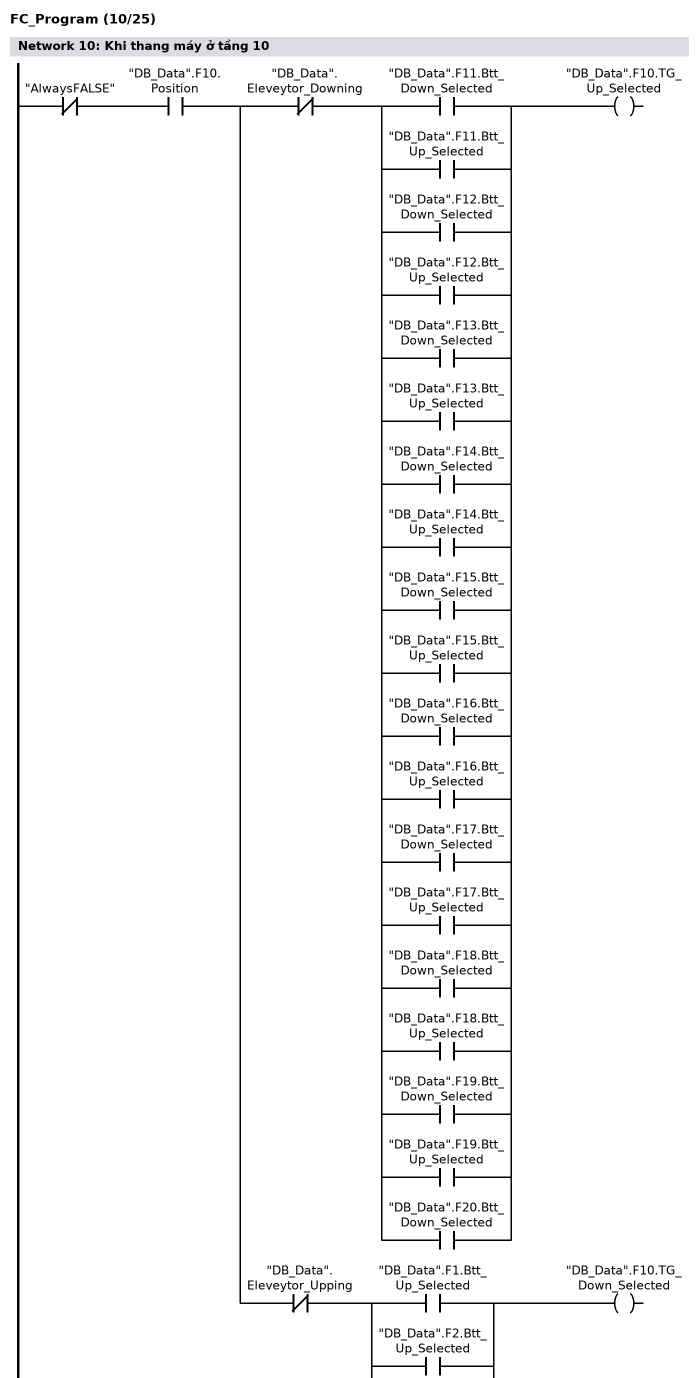
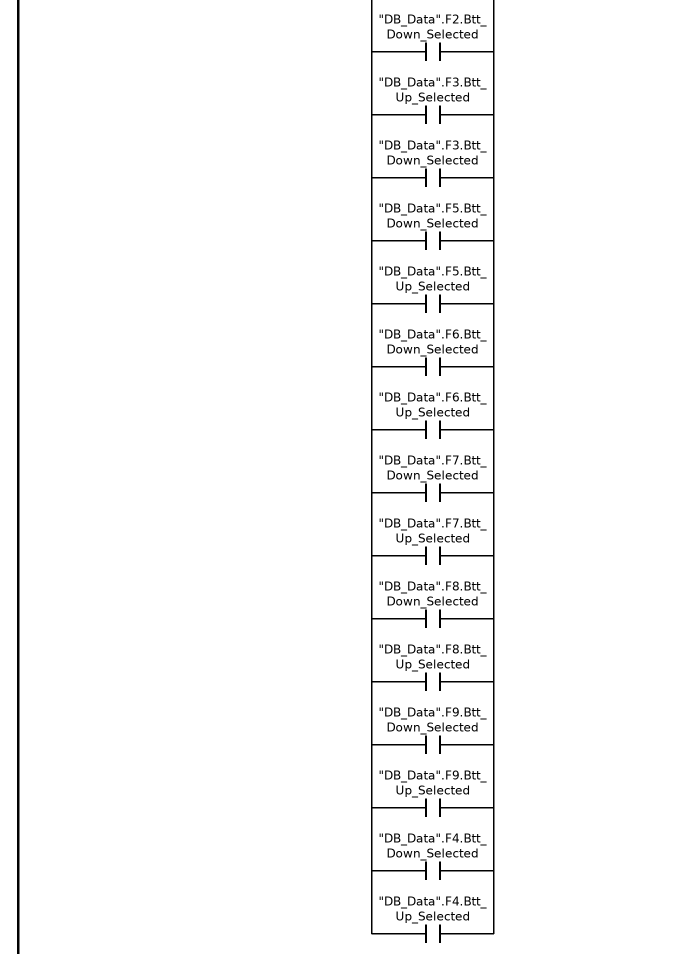
   RUNG wire#powerrail
      I_Contact( "AlwaysFALSE" )
      Contact( "DB_Data".F10.Position )
      wire#w1
      I_Contact( "DB_Data".Eleveytor_Downing )
      wire#w2
      Contact( "DB_Data".F11.Btt_Down_Selected )
      wire#w3
      Coil( "DB_Data".F10.TG_Up_Selected )
   END_RUNG
   RUNG wire#w2
      Contact( "DB_Data".F11.Btt_Up_Selected )
   END_RUNG wire#w3
   RUNG wire#w2
      Contact( "DB_Data".F12.Btt_Down_Selected )
   END_RUNG wire#w3
   RUNG wire#w2
      Contact( "DB_Data".F12.Btt_Up_Selected )
   END_RUNG wire#w3
   RUNG wire#w2
      Contact( "DB_Data".F13.Btt_Down_Selected )
   END_RUNG wire#w3
   RUNG wire#w2
      Contact( "DB_Data".F13.Btt_Up_Selected )
   END_RUNG wire#w3
   RUNG wire#w2
      Contact( "DB_Data".F14.Btt_Down_Selected )
   END_RUNG wire#w3
   RUNG wire#w2
      Contact( "DB_Data".F14.Btt_Up_Selected )
   END_RUNG wire#w3
   RUNG wire#w2
      Contact( "DB_Data".F15.Btt_Down_Selected )
   END_RUNG wire#w3
   RUNG wire#w2
      Contact( "DB_Data".F15.Btt_Up_Selected )
   END_RUNG wire#w3
   RUNG wire#w2
      Contact( "DB_Data".F16.Btt_Down_Selected )
   END_RUNG wire#w3
   RUNG wire#w2
      Contact( "DB_Data".F16.Btt_Up_Selected )
   END_RUNG wire#w3
   RUNG wire#w2
      Contact( "DB_Data".F17.Btt_Down_Selected )
   END_RUNG wire#w3
   RUNG wire#w2
      Contact( "DB_Data".F17.Btt_Up_Selected )
   END_RUNG wire#w3
   RUNG wire#w2
      Contact( "DB_Data".F18.Btt_Down_Selected )
   END_RUNG wire#w3
   RUNG wire#w2
      Contact( "DB_Data".F18.Btt_Up_Selected )
   END_RUNG wire#w3
   RUNG wire#w2
      Contact( "DB_Data".F19.Btt_Down_Selected )
   END_RUNG wire#w3
   RUNG wire#w2
      Contact( "DB_Data".F19.Btt_Up_Selected )
   END_RUNG wire#w3
   RUNG wire#w2
      Contact( "DB_Data".F20.Btt_Down_Selected )
   END_RUNG wire#w3
   RUNG wire#w1
      I_Contact( "DB_Data".Eleveytor_Upping )
      wire#w4
      Contact( "DB_Data".F1.Btt_Up_Selected )
      wire#w5
      Coil( "DB_Data".F10.TG_Down_Selected )
   END_RUNG
   RUNG wire#w4
      Contact( "DB_Data".F2.Btt_Up_Selected )
   END_RUNG wire#w5
   RUNG wire#w4
      Contact( "DB_Data".F2.Btt_Down_Selected )
   END_RUNG wire#w5
   RUNG wire#w4
      Contact( "DB_Data".F3.Btt_Up_Selected )
   END_RUNG wire#w5
   RUNG wire#w4
      Contact( "DB_Data".F3.Btt_Down_Selected )
   END_RUNG wire#w5
   RUNG wire#w4
      Contact( "DB_Data".F5.Btt_Down_Selected )
   END_RUNG wire#w5
   RUNG wire#w4
      Contact( "DB_Data".F5.Btt_Up_Selected )
   END_RUNG wire#w5
   RUNG wire#w4
      Contact( "DB_Data".F6.Btt_Down_Selected )
   END_RUNG wire#w5
   RUNG wire#w4
      Contact( "DB_Data".F6.Btt_Up_Selected )
   END_RUNG wire#w5
   RUNG wire#w4
      Contact( "DB_Data".F7.Btt_Down_Selected )
   END_RUNG wire#w5
   RUNG wire#w4
      Contact( "DB_Data".F7.Btt_Up_Selected )
   END_RUNG wire#w5
   RUNG wire#w4
      Contact( "DB_Data".F8.Btt_Down_Selected )
   END_RUNG wire#w5
   RUNG wire#w4
      Contact( "DB_Data".F8.Btt_Up_Selected )
   END_RUNG wire#w5
   RUNG wire#w4
      Contact( "DB_Data".F9.Btt_Down_Selected )
   END_RUNG wire#w5
   RUNG wire#w4
      Contact( "DB_Data".F9.Btt_Up_Selected )
   END_RUNG wire#w5
   RUNG wire#w4
      Contact( "DB_Data".F4.Btt_Down_Selected )
   END_RUNG wire#w5
   RUNG wire#w4
      Contact( "DB_Data".F4.Btt_Up_Selected )
   END_RUNG wire#w5
   // the same network as SCL:
   #_w1 := NOT "AlwaysFALSE" AND "DB_Data".F10.Position;
   "DB_Data".F10.TG_Up_Selected := #_w1 AND NOT "DB_Data".Eleveytor_Downing AND ("DB_Data".F11.Btt_Down_Selected OR "DB_Data".F11.Btt_Up_Selected OR "DB_Data".F12.Btt_Down_Selected OR "DB_Data".F12.Btt_Up_Selected OR "DB_Data".F13.Btt_Down_Selected OR "DB_Data".F13.Btt_Up_Selected OR "DB_Data".F14.Btt_Down_Selected OR "DB_Data".F14.Btt_Up_Selected OR "DB_Data".F15.Btt_Down_Selected OR "DB_Data".F15.Btt_Up_Selected OR "DB_Data".F16.Btt_Down_Selected OR "DB_Data".F16.Btt_Up_Selected OR "DB_Data".F17.Btt_Down_Selected OR "DB_Data".F17.Btt_Up_Selected OR "DB_Data".F18.Btt_Down_Selected OR "DB_Data".F18.Btt_Up_Selected OR "DB_Data".F19.Btt_Down_Selected OR "DB_Data".F19.Btt_Up_Selected OR "DB_Data".F20.Btt_Down_Selected);
   "DB_Data".F10.TG_Down_Selected := #_w1 AND NOT "DB_Data".Eleveytor_Upping AND ("DB_Data".F1.Btt_Up_Selected OR "DB_Data".F2.Btt_Up_Selected OR "DB_Data".F2.Btt_Down_Selected OR "DB_Data".F3.Btt_Up_Selected OR "DB_Data".F3.Btt_Down_Selected OR "DB_Data".F5.Btt_Down_Selected OR "DB_Data".F5.Btt_Up_Selected OR "DB_Data".F6.Btt_Down_Selected OR "DB_Data".F6.Btt_Up_Selected OR "DB_Data".F7.Btt_Down_Selected OR "DB_Data".F7.Btt_Up_Selected OR "DB_Data".F8.Btt_Down_Selected OR "DB_Data".F8.Btt_Up_Selected OR "DB_Data".F9.Btt_Down_Selected OR "DB_Data".F9.Btt_Up_Selected OR "DB_Data".F4.Btt_Down_Selected OR "DB_Data".F4.Btt_Up_Selected);
END_REGION

REGION Network 11: Khi thang máy ở tầng 11
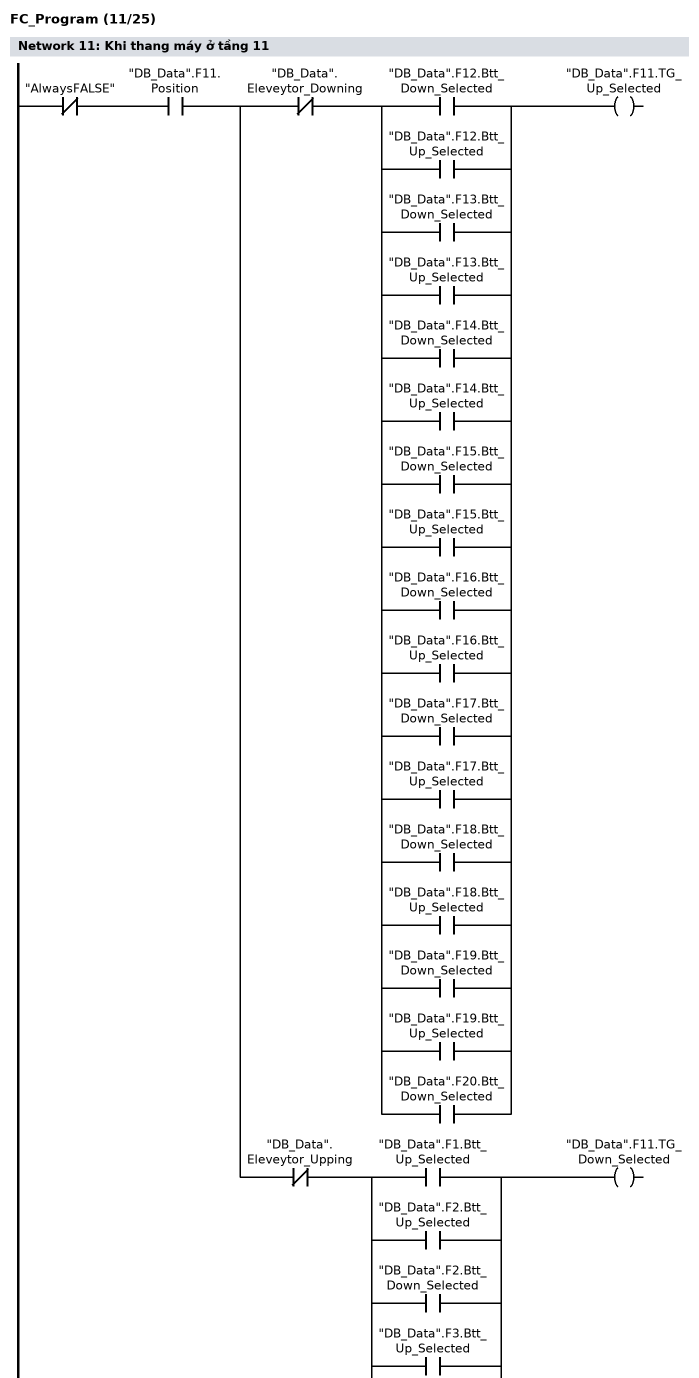
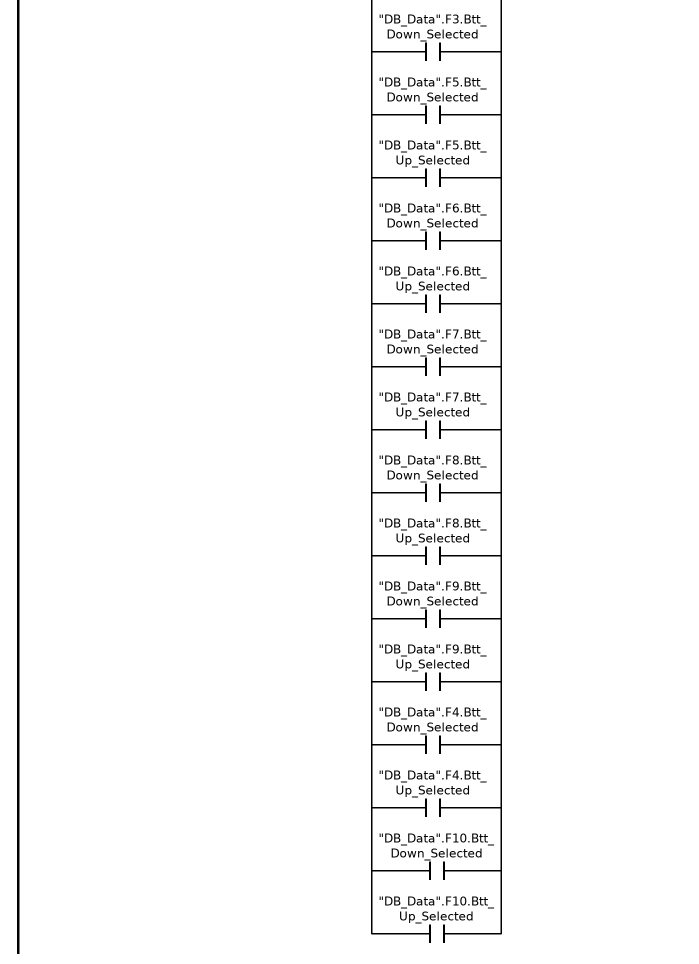
   RUNG wire#powerrail
      I_Contact( "AlwaysFALSE" )
      Contact( "DB_Data".F11.Position )
      wire#w1
      I_Contact( "DB_Data".Eleveytor_Downing )
      wire#w2
      Contact( "DB_Data".F12.Btt_Down_Selected )
      wire#w3
      Coil( "DB_Data".F11.TG_Up_Selected )
   END_RUNG
   RUNG wire#w2
      Contact( "DB_Data".F12.Btt_Up_Selected )
   END_RUNG wire#w3
   RUNG wire#w2
      Contact( "DB_Data".F13.Btt_Down_Selected )
   END_RUNG wire#w3
   RUNG wire#w2
      Contact( "DB_Data".F13.Btt_Up_Selected )
   END_RUNG wire#w3
   RUNG wire#w2
      Contact( "DB_Data".F14.Btt_Down_Selected )
   END_RUNG wire#w3
   RUNG wire#w2
      Contact( "DB_Data".F14.Btt_Up_Selected )
   END_RUNG wire#w3
   RUNG wire#w2
      Contact( "DB_Data".F15.Btt_Down_Selected )
   END_RUNG wire#w3
   RUNG wire#w2
      Contact( "DB_Data".F15.Btt_Up_Selected )
   END_RUNG wire#w3
   RUNG wire#w2
      Contact( "DB_Data".F16.Btt_Down_Selected )
   END_RUNG wire#w3
   RUNG wire#w2
      Contact( "DB_Data".F16.Btt_Up_Selected )
   END_RUNG wire#w3
   RUNG wire#w2
      Contact( "DB_Data".F17.Btt_Down_Selected )
   END_RUNG wire#w3
   RUNG wire#w2
      Contact( "DB_Data".F17.Btt_Up_Selected )
   END_RUNG wire#w3
   RUNG wire#w2
      Contact( "DB_Data".F18.Btt_Down_Selected )
   END_RUNG wire#w3
   RUNG wire#w2
      Contact( "DB_Data".F18.Btt_Up_Selected )
   END_RUNG wire#w3
   RUNG wire#w2
      Contact( "DB_Data".F19.Btt_Down_Selected )
   END_RUNG wire#w3
   RUNG wire#w2
      Contact( "DB_Data".F19.Btt_Up_Selected )
   END_RUNG wire#w3
   RUNG wire#w2
      Contact( "DB_Data".F20.Btt_Down_Selected )
   END_RUNG wire#w3
   RUNG wire#w1
      I_Contact( "DB_Data".Eleveytor_Upping )
      wire#w4
      Contact( "DB_Data".F1.Btt_Up_Selected )
      wire#w5
      Coil( "DB_Data".F11.TG_Down_Selected )
   END_RUNG
   RUNG wire#w4
      Contact( "DB_Data".F2.Btt_Up_Selected )
   END_RUNG wire#w5
   RUNG wire#w4
      Contact( "DB_Data".F2.Btt_Down_Selected )
   END_RUNG wire#w5
   RUNG wire#w4
      Contact( "DB_Data".F3.Btt_Up_Selected )
   END_RUNG wire#w5
   RUNG wire#w4
      Contact( "DB_Data".F3.Btt_Down_Selected )
   END_RUNG wire#w5
   RUNG wire#w4
      Contact( "DB_Data".F5.Btt_Down_Selected )
   END_RUNG wire#w5
   RUNG wire#w4
      Contact( "DB_Data".F5.Btt_Up_Selected )
   END_RUNG wire#w5
   RUNG wire#w4
      Contact( "DB_Data".F6.Btt_Down_Selected )
   END_RUNG wire#w5
   RUNG wire#w4
      Contact( "DB_Data".F6.Btt_Up_Selected )
   END_RUNG wire#w5
   RUNG wire#w4
      Contact( "DB_Data".F7.Btt_Down_Selected )
   END_RUNG wire#w5
   RUNG wire#w4
      Contact( "DB_Data".F7.Btt_Up_Selected )
   END_RUNG wire#w5
   RUNG wire#w4
      Contact( "DB_Data".F8.Btt_Down_Selected )
   END_RUNG wire#w5
   RUNG wire#w4
      Contact( "DB_Data".F8.Btt_Up_Selected )
   END_RUNG wire#w5
   RUNG wire#w4
      Contact( "DB_Data".F9.Btt_Down_Selected )
   END_RUNG wire#w5
   RUNG wire#w4
      Contact( "DB_Data".F9.Btt_Up_Selected )
   END_RUNG wire#w5
   RUNG wire#w4
      Contact( "DB_Data".F4.Btt_Down_Selected )
   END_RUNG wire#w5
   RUNG wire#w4
      Contact( "DB_Data".F4.Btt_Up_Selected )
   END_RUNG wire#w5
   RUNG wire#w4
      Contact( "DB_Data".F10.Btt_Down_Selected )
   END_RUNG wire#w5
   RUNG wire#w4
      Contact( "DB_Data".F10.Btt_Up_Selected )
   END_RUNG wire#w5
   // the same network as SCL:
   #_w1 := NOT "AlwaysFALSE" AND "DB_Data".F11.Position;
   "DB_Data".F11.TG_Up_Selected := #_w1 AND NOT "DB_Data".Eleveytor_Downing AND ("DB_Data".F12.Btt_Down_Selected OR "DB_Data".F12.Btt_Up_Selected OR "DB_Data".F13.Btt_Down_Selected OR "DB_Data".F13.Btt_Up_Selected OR "DB_Data".F14.Btt_Down_Selected OR "DB_Data".F14.Btt_Up_Selected OR "DB_Data".F15.Btt_Down_Selected OR "DB_Data".F15.Btt_Up_Selected OR "DB_Data".F16.Btt_Down_Selected OR "DB_Data".F16.Btt_Up_Selected OR "DB_Data".F17.Btt_Down_Selected OR "DB_Data".F17.Btt_Up_Selected OR "DB_Data".F18.Btt_Down_Selected OR "DB_Data".F18.Btt_Up_Selected OR "DB_Data".F19.Btt_Down_Selected OR "DB_Data".F19.Btt_Up_Selected OR "DB_Data".F20.Btt_Down_Selected);
   "DB_Data".F11.TG_Down_Selected := #_w1 AND NOT "DB_Data".Eleveytor_Upping AND ("DB_Data".F1.Btt_Up_Selected OR "DB_Data".F2.Btt_Up_Selected OR "DB_Data".F2.Btt_Down_Selected OR "DB_Data".F3.Btt_Up_Selected OR "DB_Data".F3.Btt_Down_Selected OR "DB_Data".F5.Btt_Down_Selected OR "DB_Data".F5.Btt_Up_Selected OR "DB_Data".F6.Btt_Down_Selected OR "DB_Data".F6.Btt_Up_Selected OR "DB_Data".F7.Btt_Down_Selected OR "DB_Data".F7.Btt_Up_Selected OR "DB_Data".F8.Btt_Down_Selected OR "DB_Data".F8.Btt_Up_Selected OR "DB_Data".F9.Btt_Down_Selected OR "DB_Data".F9.Btt_Up_Selected OR "DB_Data".F4.Btt_Down_Selected OR "DB_Data".F4.Btt_Up_Selected OR "DB_Data".F10.Btt_Down_Selected OR "DB_Data".F10.Btt_Up_Selected);
END_REGION

REGION Network 12: Khi thang máy ở tầng 12
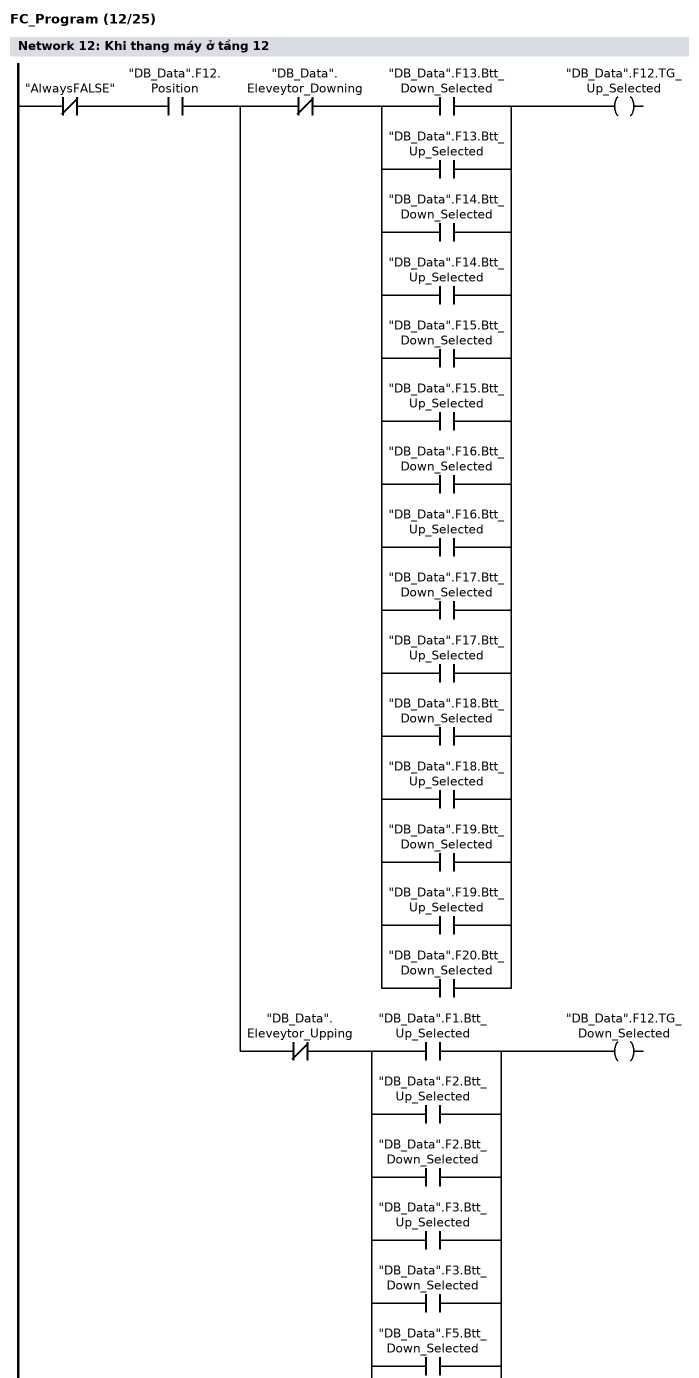
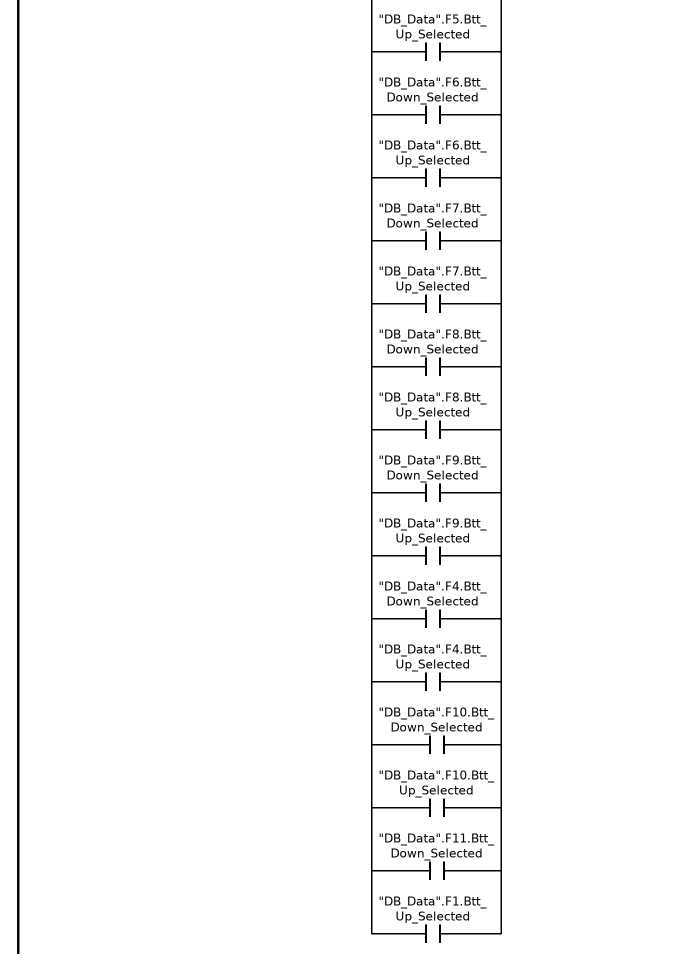
   RUNG wire#powerrail
      I_Contact( "AlwaysFALSE" )
      Contact( "DB_Data".F12.Position )
      wire#w1
      I_Contact( "DB_Data".Eleveytor_Downing )
      wire#w2
      Contact( "DB_Data".F13.Btt_Down_Selected )
      wire#w3
      Coil( "DB_Data".F12.TG_Up_Selected )
   END_RUNG
   RUNG wire#w2
      Contact( "DB_Data".F13.Btt_Up_Selected )
   END_RUNG wire#w3
   RUNG wire#w2
      Contact( "DB_Data".F14.Btt_Down_Selected )
   END_RUNG wire#w3
   RUNG wire#w2
      Contact( "DB_Data".F14.Btt_Up_Selected )
   END_RUNG wire#w3
   RUNG wire#w2
      Contact( "DB_Data".F15.Btt_Down_Selected )
   END_RUNG wire#w3
   RUNG wire#w2
      Contact( "DB_Data".F15.Btt_Up_Selected )
   END_RUNG wire#w3
   RUNG wire#w2
      Contact( "DB_Data".F16.Btt_Down_Selected )
   END_RUNG wire#w3
   RUNG wire#w2
      Contact( "DB_Data".F16.Btt_Up_Selected )
   END_RUNG wire#w3
   RUNG wire#w2
      Contact( "DB_Data".F17.Btt_Down_Selected )
   END_RUNG wire#w3
   RUNG wire#w2
      Contact( "DB_Data".F17.Btt_Up_Selected )
   END_RUNG wire#w3
   RUNG wire#w2
      Contact( "DB_Data".F18.Btt_Down_Selected )
   END_RUNG wire#w3
   RUNG wire#w2
      Contact( "DB_Data".F18.Btt_Up_Selected )
   END_RUNG wire#w3
   RUNG wire#w2
      Contact( "DB_Data".F19.Btt_Down_Selected )
   END_RUNG wire#w3
   RUNG wire#w2
      Contact( "DB_Data".F19.Btt_Up_Selected )
   END_RUNG wire#w3
   RUNG wire#w2
      Contact( "DB_Data".F20.Btt_Down_Selected )
   END_RUNG wire#w3
   RUNG wire#w1
      I_Contact( "DB_Data".Eleveytor_Upping )
      wire#w4
      Contact( "DB_Data".F1.Btt_Up_Selected )
      wire#w5
      Coil( "DB_Data".F12.TG_Down_Selected )
   END_RUNG
   RUNG wire#w4
      Contact( "DB_Data".F2.Btt_Up_Selected )
   END_RUNG wire#w5
   RUNG wire#w4
      Contact( "DB_Data".F2.Btt_Down_Selected )
   END_RUNG wire#w5
   RUNG wire#w4
      Contact( "DB_Data".F3.Btt_Up_Selected )
   END_RUNG wire#w5
   RUNG wire#w4
      Contact( "DB_Data".F3.Btt_Down_Selected )
   END_RUNG wire#w5
   RUNG wire#w4
      Contact( "DB_Data".F5.Btt_Down_Selected )
   END_RUNG wire#w5
   RUNG wire#w4
      Contact( "DB_Data".F5.Btt_Up_Selected )
   END_RUNG wire#w5
   RUNG wire#w4
      Contact( "DB_Data".F6.Btt_Down_Selected )
   END_RUNG wire#w5
   RUNG wire#w4
      Contact( "DB_Data".F6.Btt_Up_Selected )
   END_RUNG wire#w5
   RUNG wire#w4
      Contact( "DB_Data".F7.Btt_Down_Selected )
   END_RUNG wire#w5
   RUNG wire#w4
      Contact( "DB_Data".F7.Btt_Up_Selected )
   END_RUNG wire#w5
   RUNG wire#w4
      Contact( "DB_Data".F8.Btt_Down_Selected )
   END_RUNG wire#w5
   RUNG wire#w4
      Contact( "DB_Data".F8.Btt_Up_Selected )
   END_RUNG wire#w5
   RUNG wire#w4
      Contact( "DB_Data".F9.Btt_Down_Selected )
   END_RUNG wire#w5
   RUNG wire#w4
      Contact( "DB_Data".F9.Btt_Up_Selected )
   END_RUNG wire#w5
   RUNG wire#w4
      Contact( "DB_Data".F4.Btt_Down_Selected )
   END_RUNG wire#w5
   RUNG wire#w4
      Contact( "DB_Data".F4.Btt_Up_Selected )
   END_RUNG wire#w5
   RUNG wire#w4
      Contact( "DB_Data".F10.Btt_Down_Selected )
   END_RUNG wire#w5
   RUNG wire#w4
      Contact( "DB_Data".F10.Btt_Up_Selected )
   END_RUNG wire#w5
   RUNG wire#w4
      Contact( "DB_Data".F11.Btt_Down_Selected )
   END_RUNG wire#w5
   RUNG wire#w4
      Contact( "DB_Data".F1.Btt_Up_Selected )
   END_RUNG wire#w5
   // the same network as SCL:
   #_w1 := NOT "AlwaysFALSE" AND "DB_Data".F12.Position;
   "DB_Data".F12.TG_Up_Selected := #_w1 AND NOT "DB_Data".Eleveytor_Downing AND ("DB_Data".F13.Btt_Down_Selected OR "DB_Data".F13.Btt_Up_Selected OR "DB_Data".F14.Btt_Down_Selected OR "DB_Data".F14.Btt_Up_Selected OR "DB_Data".F15.Btt_Down_Selected OR "DB_Data".F15.Btt_Up_Selected OR "DB_Data".F16.Btt_Down_Selected OR "DB_Data".F16.Btt_Up_Selected OR "DB_Data".F17.Btt_Down_Selected OR "DB_Data".F17.Btt_Up_Selected OR "DB_Data".F18.Btt_Down_Selected OR "DB_Data".F18.Btt_Up_Selected OR "DB_Data".F19.Btt_Down_Selected OR "DB_Data".F19.Btt_Up_Selected OR "DB_Data".F20.Btt_Down_Selected);
   "DB_Data".F12.TG_Down_Selected := #_w1 AND NOT "DB_Data".Eleveytor_Upping AND ("DB_Data".F1.Btt_Up_Selected OR "DB_Data".F2.Btt_Up_Selected OR "DB_Data".F2.Btt_Down_Selected OR "DB_Data".F3.Btt_Up_Selected OR "DB_Data".F3.Btt_Down_Selected OR "DB_Data".F5.Btt_Down_Selected OR "DB_Data".F5.Btt_Up_Selected OR "DB_Data".F6.Btt_Down_Selected OR "DB_Data".F6.Btt_Up_Selected OR "DB_Data".F7.Btt_Down_Selected OR "DB_Data".F7.Btt_Up_Selected OR "DB_Data".F8.Btt_Down_Selected OR "DB_Data".F8.Btt_Up_Selected OR "DB_Data".F9.Btt_Down_Selected OR "DB_Data".F9.Btt_Up_Selected OR "DB_Data".F4.Btt_Down_Selected OR "DB_Data".F4.Btt_Up_Selected OR "DB_Data".F10.Btt_Down_Selected OR "DB_Data".F10.Btt_Up_Selected OR "DB_Data".F11.Btt_Down_Selected OR "DB_Data".F1.Btt_Up_Selected);
END_REGION

REGION Network 13: Khi thang máy ở tầng 13
